	IF Modbus_Slave.rBias_2>rStepBias THEN
		rStepBias:=rStepBias+rStep;
		IF rStepBias>=Modbus_Slave.rBias_2 THEN
			rStepBias:=Modbus_Slave.rBias_2;
		END_IF
	ELSIF Modbus_Slave.rBias_2<rStepBias THEN
		rStepBias:=rStepBias-rStep;
		IF rStepBias<=Modbus_Slave.rBias_2 THEN
			rStepBias:=Modbus_Slave.rBias_2;
		END_IF
	END_IF
	rAuToStepBiasTemp:=0;
ELSIF GVL.bStartTrack AND Axis2Remote.iMode=2 THEN
	Axis2Remote.bStartAutoTrack := TRUE;
	Axis2Remote.rChanU := -AutoTrackingCal.rChanUa;
ELSE
	Axis2Remote.bStartAutoTrack := FALSE;	
	rAuToStepBias:=0;
	rStepBias:=0;
	rAuToStepBiasTemp:=0;
END_IF

// 本控自跟踪
IF GVL.bStartLocalAutoTrack AND Axis2Local.iMode = 4 THEN
	Axis2Local.bStartAutoTrack := TRUE;
	Axis2Local.rChanU := -AutoTrackingCal.rChanUaLocal;
ELSE
	Axis2Local.bStartAutoTrack := FALSE;
END_IF

// =============================================================================
// 段 9: 合成 rPIDCmdPos（注意 AZ_out 为减）→ Az_Ctrl_FB
// =============================================================================
Axis2Remote.rPIDCmdPos:=RealTimePosCal.rInterAzPos+rStepBias+rAuToStepBias+rSearchNextStepTarget-SECURITYCHECK.AZ_out+rAuToStepBiasTemp;

IF Axis2Remote.rPIDCmdPos<-275 THEN
	Axis2Remote.rPIDCmdPos:=-275;
ELSIF Axis2Remote.rPIDCmdPos>275 THEN
	Axis2Remote.rPIDCmdPos:=275;
END_IF

Axis2_Ctrl(sLocal:=Axis2Local, sCtrl:=Axis2Remote, sStatus:=Axis2Status, sVisible:=Axis2Visible, rRealPos:=rFctPosReal_2, rPosLimK:=0.34);

END_PROGRAM

// Device/Application/El_ctrl_1
PROGRAM El_ctrl_1

VAR
    Axis1_Ctrl : El_Ctrl_FB;           // 俯仰轴控制 FB（阶段 4 已注释）
    bRemote2LocalStop : BOOL;          // 远控→本控切换中，需先减速下电
    bLocal2RemoteStop : BOOL;          // 本控→远控切换中，需先减速下电
    Error : INT;                       // 保留
    Axis1Limit_pos : REAL;             // 硬限位上限 180°
    Axis1Limit_Neg : REAL;             // 硬限位下限 93°
    bRTriger : Standard.R_TRIG;        // bLocalCtrl 上升沿（切到本控）
    bFTriger : Standard.F_TRIG;        // bLocalCtrl 下降沿（切到远控）
    Stop1_Count : INT;                 // 低速持续计数（用于判定已停稳）
    bStop_1 : BOOL;                    // TRUE=俯仰轴已停稳（|v|<0.035 持续>1s）
    rPosModeStepBias : LREAL;          // 保留/指向模式步进偏置
    rPosModeStep : LREAL;
    rStepBiasMax : LREAL;
    rStepBias : LREAL;                 // Modbus 下发的手动偏置，逐步逼近 rBias_1
    rStep : LREAL;                     // rStepBias 每拍变化步长
    rAuToStepBias : LREAL;             // 自跟踪累积拉偏 (deg)
    rAuToStepBiasTemp : LREAL;         // 自跟踪瞬时拉偏分量
    rAutoStep : LREAL;                 // 关闭自跟踪后 rAuToStepBias 归零步长
    TbAutoTrigger : Standard.F_TRIG;
    RbAutoTrigger : Standard.R_TRIG;
    rAutoTrackingBiasMax : LREAL;      // 自跟踪拉偏上限
    rLocalInitPosModeSpeed : REAL;
    rRemoteInitPosModeSpeed : REAL;
    iCountOffAuto : INT;
    iCasePBAutoTrack : INT;
    rKAuToStepBias : LREAL;            // 自跟踪拉偏增益系数
    agcmaxsearch_tb : AGCMaxSearch_PB_1;  // 指向模式(mode2) AGC 峰值搜索
    rSearchNextStepTarget_tb : REAL;      // 指向模式搜索输出偏置
    agcmaxsearch_pb : AGCMaxSearch_PB_1;  // 程引模式(mode4) AGC 峰值搜索
    rElthreshold : REAL;               // 俯仰角阈值：仅高于此值才在程引下做 AGC 搜索
    toN1 : Standard.Ton;
    ttime1 : TIME;
    bstartagcmaxsearch : BOOL;
    rSearchNextStepTarget : REAL;      // 程引模式 AGC 搜索输出偏置
    rMaxPosTest : REAL;                // AGC 搜索调试：峰值位置
END_VAR


(*==============================================================================
  PRG: El_ctrl_1（俯仰轴 El 顶层程序）
  任务: Canopen 10ms
  作用:
    1. 读 CANopen 反馈 → 换算实际速度/位置 (rFctVelReal_1 / rFctPosReal_1)
    2. 组装 Axis1Status（故障、使能、运动中等）
    3. 远/本控切换保护、自跟踪拉偏、AGC 峰值搜索
    4. 合成 PID 目标位置 rPIDCmdPos → 调用 El_Ctrl_FB
  数据流:
    Modbus/上位机 → Axis1Remote（在 Modbus_Slave 等处赋值）
    RealTimePosCal.rInterElPos + 各类偏置 → rPIDCmdPos → El_Ctrl_FB → GVL.diEl*
==============================================================================*)




(* 远控参量曾在此从 Modbus_Slave 直赋，现改由 Modbus_Slave 程序统一写入 Axis1Remote *)

// =============================================================================
// 段 1: 驱动状态字 → Axis1Status（供 El_Ctrl_FB 与 HMI 使用）
// DS402 状态: bit0/1/2 同时为 1 表示 Operation Enabled（伺服已使能）
// =============================================================================
Axis1Status.Error := GVL.bElStsBit3;
Axis1Status.ErrorID := GVL.eElErrorcode;
Axis1Status.bServo_Enable := GVL.bElStsBit0 AND GVL.bElStsBit1 AND GVL.bElStsBit2;
Axis1Status.bBrake := NOT (GVL.bElStsBit0 AND GVL.bElStsBit1 AND GVL.bElStsBit2);
Axis1Status.Disabled := NOT (GVL.bElStsBit0 AND GVL.bElStsBit1 AND GVL.bElStsBit2);
// 软限位写入命令结构体（与下面硬限位 93~180 一致）
Axis1Remote.rSoft_limit_Negative:=93;Axis1Remote.rSoft_limit_Postive:=180;
Axis1Local.rSoft_limit_Negative:=93;Axis1Local.rSoft_limit_Postive:=180;

// =============================================================================
// 段 2: CANopen 反馈 → 实际速度/位置（deg, deg/s）
// 公式: 物理量 = diActXxx / 524288 × 360；俯仰另加 Modbus 标定偏移 lrElOffset
// =============================================================================
rFctVelReal_1:=DINT_TO_REAL(diElActVel)/524288.0*360.0;
rFctPosReal_1:=DINT_TO_REAL(diElActPos)/524288.0*360.0 + modbus_slave.lrElOffset;

// =============================================================================
// 段 3: 指向命令硬限位（远控/本控 rPosCmd 钳位到 93°~180°）
// =============================================================================
Axis1Limit_pos:=180;
Axis1Limit_Neg:=93;
IF Axis1Remote.rPosCmd>Axis1Limit_pos THEN
	Axis1Remote.rPosCmd:=180;
ELSIF Axis1Remote.rPosCmd<Axis1Limit_Neg THEN
	 Axis1Remote.rPosCmd:=93;  
END_IF

IF Axis1Local.rPosCmd>Axis1Limit_pos THEN
	Axis1Local.rPosCmd:=180;
ELSIF Axis1Local.rPosCmd<Axis1Limit_Neg THEN
	 Axis1Local.rPosCmd:=93;  
END_IF

// =============================================================================
// 段 4: 停稳判定 → Axis1Status.Moving
// |速度|<0.035°/s 连续 100 拍(约1s) 认为停稳；bStop_1=TRUE → Moving=FALSE
// =============================================================================
IF  ABS(rFctVelReal_1)<0.035 THEN
	Stop1_Count:=Stop1_Count+1;
	IF Stop1_Count>100 THEN
		Stop1_Count:=101;
		bStop_1:=TRUE;;
	END_IF
ELSE
	Stop1_Count:=0;
	bStop_1:=FALSE;
END_IF
Axis1Status.Moving := NOT bStop_1;

// =============================================================================
// 段 5: PID 使能 — 仅指向(2)与程引(4)模式需要位置环
// =============================================================================
IF Axis1Remote.iMode=2 OR Axis1Remote.iMode=4 THEN
	Axis1Remote.bPIDEnable:=TRUE;
ELSE
	Axis1Remote.bPIDEnable:=FALSE;
END_IF

// =============================================================================
// 段 6: 远控 ↔ 本控 切换保护（GVL.bLocalCtrl）
// 切换瞬间若伺服仍使能 → 置切换标志 → 强制 mode=7(halt) 减速
// 停稳且下电完成后 → mode=0，清除标志
// =============================================================================
bRTriger(CLK:=GVL.bLocalCtrl);
bFTriger(CLK:=GVL.bLocalCtrl);

// 远控 → 本控（bLocalCtrl 上升沿）
IF Axis1Status.bServo_Enable AND (bRTriger.Q ) THEN//如果速度不为0且本控发生切换，则减速停止标识为True
	bRemote2LocalStop:=TRUE;
END_IF
IF bRemote2LocalStop  THEN //若减速停止标识符为True 
	
	IF  bStop_1=TRUE THEN//且电机速度不为0 开始减速 减速完成后下使能，下使能完成后复位标识符复位
		Axis1Local.iMode:=0;
		Axis1Remote.iMode:=0;
		IF Axis1Status.bServo_Enable=FALSE THEN
			bRemote2LocalStop:=FALSE;
		END_IF
	ELSE
		Axis1Local.iMode:=7;
		Axis1Remote.iMode:=7;
	END_IF
END_IF

// 本控 → 远控（bLocalCtrl 下降沿）
IF Axis1Status.bServo_Enable AND (bFTriger.Q ) THEN//如果速度不为0且本控发生切换，则减速停止标识为True
	bLocal2RemoteStop:=TRUE;
END_IF
IF bLocal2RemoteStop  THEN //若减速停止标识符为True 
	
	IF  bStop_1=TRUE THEN//且电机速度不为0 开始减速 减速完成后下使能，下使能完成后复位标识符复位
		Axis1Local.iMode:=0;
		Axis1Remote.iMode:=0;
		IF Axis1Status.bServo_Enable=FALSE THEN
			bLocal2RemoteStop:=FALSE;
		END_IF
	ELSE
		Axis1Remote.iMode:=7;
		Axis1Local.iMode:=7;
	END_IF
END_IF

// =============================================================================
// 段 7: AGC 峰值搜索（与方位 Az_ctrl_1 协同，bstartSearchEl 由方位触发）
// mode2: 插值目标 = rPosCmd；mode4: 插值目标 = RealTimePosCal.rInterElPos
// 仅当俯仰高于 rElthreshold（相对水平）且在程引下才在 mode4 启用搜索
// =============================================================================
IF Axis1Remote.iMode=2 THEN
			IF GVL.Chan1AGC>=(GVL.Chanthreshold-0.1) THEN
					agcmaxsearch_pb(bstart:=Az_ctrl_1.agcmaxsearch_tb.bSucess,rAGCNow:=GVL.Chan1AGC,btrig:=Az_ctrl_1.bstartSearchEl,
						rCurrentPos:=rFctPosReal_1,rInterPos:=Axis1Remote.rPosCmd,
				rStepBiasNow:=rStepBias,bAutoTracking:=GVL.bStartTrack,bStop:=FALSE,
				rStepBias=>rSearchNextStepTarget_tb,rAGCMaxBias=>rMaxPosTest,bSucess=>);
			ELSE
				bstartagcmaxsearch:=FALSE;
				agcmaxsearch_pb(bstart:=Az_ctrl_1.agcmaxsearch_tb.bSucess,rAGCNow:=GVL.Chan1AGC,btrig:=Az_ctrl_1.bstartSearchEl,
				rCurrentPos:=rFctPosReal_1,rInterPos:=Axis1Remote.rPosCmd,
				rStepBiasNow:=rStepBias,bAutoTracking:=GVL.bStartTrack,bStop:=FALSE,
				rStepBias=>rSearchNextStepTarget_tb,rAGCMaxBias=>rMaxPosTest,bSucess=>);
			END_IF
		ELSIF Axis1Remote.iMode=4 AND rFctPosReal_1-90>rElthreshold  THEN
			IF GVL.Chan1AGC>=(GVL.Chanthreshold-0.1) THEN
					agcmaxsearch_pb(bstart:=Az_ctrl_1.agcmaxsearch_pb.bSucess,rAGCNow:=GVL.Chan1AGC,btrig:=Az_ctrl_1.bstartSearchEl,
						rCurrentPos:=rFctPosReal_1,rInterPos:=RealTimePosCal.rInterElPos,
				rStepBiasNow:=rStepBias,bAutoTracking:=GVL.bStartTrack,bStop:=FALSE,
				rStepBias=>rSearchNextStepTarget,rAGCMaxBias=>rMaxPosTest,bSucess=>);
			ELSE
				bstartagcmaxsearch:=FALSE;
				agcmaxsearch_pb(bstart:=Az_ctrl_1.agcmaxsearch_pb.bSucess,rAGCNow:=GVL.Chan1AGC,btrig:=Az_ctrl_1.bstartSearchEl,
				rCurrentPos:=rFctPosReal_1,rInterPos:=RealTimePosCal.rInterElPos,
				rStepBiasNow:=rStepBias,bAutoTracking:=GVL.bStartTrack,bStop:=FALSE,
				rStepBias=>rSearchNextStepTarget,rAGCMaxBias=>rMaxPosTest,bSucess=>);
			END_IF
		ELSIF Axis1Remote.iMode =0  OR Axis1Remote.iMode =7 THEN
			bstartagcmaxsearch:=FALSE;
			agcmaxsearch_pb(bstart:=Az_ctrl_1.agcmaxsearch_pb.bSucess,rAGCNow:=GVL.Chan1AGC,btrig:=Az_ctrl_1.bstartSearchEl,
			rCurrentPos:=rFctPosReal_1,rInterPos:=RealTimePosCal.rInterElPos,	
			rStepBiasNow:=rStepBias,bAutoTracking:=GVL.bStartTrack,bStop:=FALSE,
			rStepBias=>rSearchNextStepTarget,rAGCMaxBias=>rMaxPosTest,bSucess=>);
		END_IF

// =============================================================================
// 段 8: 自跟踪拉偏（远控）
// mode4+程引: 用 AutoTrackingCal.rChanUe 累积 rAuToStepBias（限幅）
// mode2+指向: 直接用 rChanU 作 PID 目标增量（在 El_Ctrl_FB 内 rChanU+位置）
// 关跟踪: rAuToStepBias 渐零，rStepBias 渐近 Modbus_Slave.rBias_1
// =============================================================================
IF GVL.bStartTrack AND Axis1Remote.iMode=4 THEN
	Axis1Remote.bStartAutoTrack := TRUE;
	IF rAuToStepBias > rAutoTrackingBiasMax THEN
		rAuToStepBias := rAutoTrackingBiasMax;
	ELSIF rAuToStepBias < -rAutoTrackingBiasMax THEN
		rAuToStepBias := -rAutoTrackingBiasMax;
	ELSE
		rAuToStepBiasTemp:=0.02*AutoTrackingCal.rDirSenFac*AutoTrackingCal.rChanUe;
		rAuToStepBias:=rAuToStepBias+AutoTrackingCal.rDirSenFac*rKAuToStepBias*AutoTrackingCal.rChanUe/1000.0;
	END_IF
ELSIF NOT GVL.bStartTrack AND Axis1Remote.iMode=4 THEN
	IF 	rAuToStepBias>0 THEN//关闭自跟踪后自跟踪拉偏量逐渐归0
		rAuToStepBias:=rAuToStepBias-rAutoStep;
	ELSIF rAuToStepBias<0 THEN
		rAuToStepBias:=rAuToStepBias+rAutoStep;
	ELSE
		rAuToStepBias:=0;
	END_IF
	
	IF Modbus_Slave.rBias_1>rStepBias THEN
		rStepBias:=rStepBias+rStep;
		IF rStepBias>=Modbus_Slave.rBias_1 THEN
			rStepBias:=Modbus_Slave.rBias_1;
		END_IF
	ELSIF Modbus_Slave.rBias_1<rStepBias THEN
		rStepBias:=rStepBias-rStep;
		IF rStepBias<=Modbus_Slave.rBias_1 THEN
			rStepBias:=Modbus_Slave.rBias_1;
		END_IF
	END_IF
	rAuToStepBiasTemp:=0;
ELSIF GVL.bStartTrack AND Axis1Remote.iMode=2 THEN
	Axis1Remote.bStartAutoTrack := TRUE;
	Axis1Remote.rChanU := AutoTrackingCal.rChanUe;
ELSE
	Axis1Remote.bStartAutoTrack := FALSE;	
	rAuToStepBias:=0;
	rStepBias:=0;
	rAuToStepBiasTemp:=0;
END_IF

// 本控自跟踪（仅程引 mode4）
IF GVL.bStartLocalAutoTrack AND Axis1Local.iMode = 4 THEN
	Axis1Local.bStartAutoTrack := TRUE;
	Axis1Local.rChanU := AutoTrackingCal.rChanUeLocal;
ELSE
	Axis1Local.bStartAutoTrack := FALSE;
END_IF

// =============================================================================
// 段 9: 合成 PID 目标位置并限位 → 调用 El_Ctrl_FB
// rPIDCmdPos = 程引插值 + 手动偏置 + 自跟踪偏置 + AGC搜索偏置 + 安全检查偏置
// =============================================================================
Axis1Remote.rPIDCmdPos:=RealTimePosCal.rInterElPos+rStepBias+rAuToStepBias+rSearchNextStepTarget+SECURITYCHECK.el_out+rAuToStepBiasTemp;
IF Axis1Remote.rPIDCmdPos<93 THEN
	Axis1Remote.rPIDCmdPos:=93;
ELSIF Axis1Remote.rPIDCmdPos>180 THEN
	Axis1Remote.rPIDCmdPos:=180;
END_IF

Axis1_Ctrl(sLocal:=Axis1Local, sCtrl:=Axis1Remote, sStatus:=Axis1Status, sVisible:=Axis1Visible, rRealPos:=rFctPosReal_1, rPosLimK:=0.34);

END_PROGRAM

// Device/Application/PID
FUNCTION_BLOCK PID
VAR_INPUT
    rTarget : REAL;              // 目标位置 (deg)
    rFeedback : REAL;            // 实际位置反馈 (deg)
    rPosLimPositive : LREAL;     // 软限位正限 (deg)，超出则输出清零
    rPosLimNegative : LREAL;     // 软限位负限 (deg)
    rKp : REAL;                  // 比例系数
    rKi : REAL;                  // 积分系数
    rKd : REAL;                  // 微分系数（当前逻辑未实际使用）
    iThreshold : INT;            // 积分开启阈值 (deg)；-1 = 始终开积分
    bPIDEnable : BOOL;           // PID 使能，FALSE 时各项清零
    rVelLim : LREAL;             // 输出速度限幅 (deg/s)
END_VAR

VAR_OUTPUT
    rPIDOutput : LREAL;          // PID 输出速度 (deg/s)，写到 diXxTargetVel 前换算
    rPIDtrace : LREAL;           // 调试/显示用，与 rPIDOutput 相同
END_VAR
VAR
    rLastError : LREAL;          // 上一拍误差（当前版本未使用微分，保留备用）
    rErrorNow : LREAL;           // 当前误差 = rTarget - rFeedback
    rIntegralNew : LREAL;        // 积分累计量
    rDerivativeNew : LREAL;      // 微分项（未使用）
    rDelta : LREAL;              // 备用
    rProportionNew : LREAL;      // 比例项 = rErrorNow
END_VAR


(*==============================================================================
  FB: PID（位置环速度输出 PID）
  任务: Canopen 10ms（由 *_Ctrl_FB 调用）
  作用: 输入目标位置与实际位置，输出速度指令（deg/s）
  算法: 比例 + 条件积分（误差小于阈值才累积），无微分
  使用者: El_Ctrl_FB / Az_Ctrl_FB / Ti_Ctrl_FB 中的 VelPID_1/2/3
==============================================================================*)

// ----- 段：PID 使能入口 -----
IF (bPIDEnable>0) THEN //如果PID使能
	IF rTarget=rFeedback THEN
		rPIDOutput:=0;	               // 目标=反馈，输出为 0
	ELSE
	
		rErrorNow:=rTarget-rFeedback;  //计算当前误差 en
		rProportionNew:=rErrorNow;     //比例项

		// ----- 段：条件积分（仅在软限位内、误差小于阈值时才累积）-----
		IF rFeedback>rPosLimNegative AND rFeedback<rPosLimPositive THEN //若在软限位之内，工作时开启积分项
			IF (ABS(rTarget-rFeedback)<iThreshold) THEN//位置差小于积分阈值
				rIntegralNew:= rIntegralNew+rErrorNow; //积分项
			ELSE
				rIntegralNew:=0;
			END_IF;
		ELSE //不在软限位范围内,则积分项为0
			rIntegralNew:=0;
		END_IF

		// ----- 段：PID 求和输出 -----
		rPIDOutPut:=rKp*rProportionNew+rKi*rIntegralNew;
		rPIDtrace:=rKp*rProportionNew+rKi*rIntegralNew;

		// ----- 段：速度限幅（双向） -----
		IF rPIDOutput<(-rVelLim) THEN
			rPIDOutput:=-rVelLim;
		ELSIF rPIDOutput>rVelLim THEN
			rPIDOutput:=rVelLim;
		END_IF
		
		// ----- 段：超软限位时强制输出清零，防止继续向限位方向运动 -----
		IF rFeedback>rPosLimPositive AND rPIDOutput>0 THEN 
			rPIDOutput:=0;
		END_IF
		IF rFeedback<rPosLimNegative AND rPIDOutput<0 THEN
			rPIDOutput:=0;
		END_IF
		
		rLastError:=rErrorNow;//将当前误差赋值给上一次误差
		
	END_IF
ELSE//非使能清零PID各项
	rProportionNew:=0.0;
	rIntegralNew:=0.0;
	rPIDOutput:=0.0;
END_IF

END_FUNCTION_BLOCK

// Device/Application/El_Ctrl_FB
FUNCTION_BLOCK El_Ctrl_FB

VAR_INPUT
    sLocal : AxisCrtlStruct;     // 本控命令结构体（来自本地操作面板/GVL.sXxLocal）
    sCtrl : AxisCrtlStruct;      // 远控命令结构体（来自 Modbus/上位机/GVL.sXxCtrl）
    sStatus : AxisStatus;        // 轴状态（Disabled/Moving/Error 等标志）
    sVisible : AxisVisible;      // HMI 可视化相关（此 FB 内部未直接使用）
    rRealPos : REAL;             // 编码器实际位置 (deg)，即 GVL.rFctPosReal_X
    rPosLimK : REAL;             // 备用限位系数（当前逻辑未使用）
END_VAR

VAR_OUTPUT
    logicError : INT;            // 逻辑错误码（保留，当前未赋值）
END_VAR

VAR
    VelPID_1 : PID;              // 位置模式（positionMode）用普通 PID
    VelPID_2 : PID;              // 本控位置模式（programBootMode 本控）用普通 PID
    VelPID_3 : PID;              // 保留（已被 vpid1 替代，代码中注释掉）
    vpid1 : vpid;                // 变增益 PID，用于 programBootMode 远控/自跟踪
    TON_0 : TON;                 // 延时 1s，错误时判断 stop0 是否超时
    bTick : BOOL;                // stop0 超时后置位，触发强制下电
    tr : BOOL;                   // 心跳错误正在处理中标志（防止重入）
    icount1 : INT;               // 心跳恢复计数器（等 101 拍 ≈ 1s 后清 bit7）
    icount2 : INT;               // 清 bit7 后再等 101 拍才结束保护
    icount3 : INT;               // 备用
    bfin1 : BOOL;                // icount1 到达后置位，触发 icount2 阶段
    bfin2 : BOOL;                // 保留
    istate : INT;                // 上电序列状态机（0→1→2）
    icount : INT;                // 上电序列各步骤等待计数（20 拍 = 200ms）
END_VAR


(*==============================================================================
  FB: El_Ctrl_FB（俯仰轴 Elevation 控制功能块）
  任务: Canopen 10ms（周期调用）
  作用:
    - 根据 sCtrl/sLocal 的 iMode，产生对应 CANopen 速度/控制字写入
    - 封装上/下电序列、软限位保护、CANopen 错误码自动恢复、心跳丢失处理
    - 内部调用 PID / vpid 进行位置→速度的闭环换算
  输入: sCtrl（远控命令结构体）、sLocal（本控命令结构体）
        sStatus（轴状态）、rRealPos（编码器实际角度）
  输出: 直接写 GVL.diElTargetVel / diElTargetAcc / diElTargetDec 及控制字位

  速度换算公式（通用）:
    diXxTargetVel [inc/s] = deg/s × 524288 / 360
    其中 524288 = 2^19（CANopen 电机编码器增量/转，具体由电机参数决定）
==============================================================================*)


// =============================================================================
// 段 A: 全局复位 — 轴停止或下电时清 bit8（快速停止位）
// bit8=1 激活快速停止，bit8=0 正常运行
// =============================================================================
IF sStatus.Disabled OR (NOT sStatus.Moving) THEN
	bElCtrlBit8 := FALSE;
END_IF

// =============================================================================
// 段 B: 错误复位（由 HMI 或 Modbus 写 bError_Reset）
// 将两个命令结构体模式设为 reset(6)，清 Error_code
// =============================================================================
IF GVL.bError_Reset THEN
	sCtrl.iMode:=6;
	sLocal.iMode:=6;
	GVL.Error_code:=0;
END_IF
IF GVL.Error_code =0 THEN
	GVL.bError_Reset:=FALSE;
END_IF

// =============================================================================
// 段 C: CANopen 心跳超时错误（错误码 0x8130）自动恢复序列
// 步骤: 设 bit7(故障复位位) → 等 101 拍 → 清 bit7 → 再等 101 拍 → 结束
// 期间同时下电（清控制字 bit0~3），待驱动自愈后再由上层重新上电
// =============================================================================
IF GVL.eElErrorcode = 16#8130 AND NOT tr THEN
	GVL.bElCtrlBit7 := TRUE;  // 触发驱动故障复位
	tr:=TRUE;
	istate:=0;
	icount:=0;
	// 写入下电控制字
	GVL.bElCtrlBit3 := FALSE;
	GVL.bElCtrlBit0 := FALSE;
	GVL.bElCtrlBit1 := FALSE;
	GVL.bElCtrlBit2 := FALSE;	
END_IF
IF tr THEN
	icount1 := icount1 + 1;
END_IF
IF icount1 > 101 THEN     // 约 1s（10ms × 101）后清故障复位位
	icount1 := 0;
	tr := FALSE;
	GVL.bElCtrlBit7 := FALSE;
	bfin1 := TRUE;
END_IF
IF bfin1 THEN             // 再等 1s 让驱动彻底稳定
	icount2 := icount2 + 1;
END_IF
IF icount2 > 101 THEN
	bfin1 := FALSE;
	icount2 := 0;
END_IF

// =============================================================================
// 段 D: 主控制逻辑
// 条件: 无全局错误 AND 无驱动错误 AND 不在心跳恢复序列中
// =============================================================================
IF GVL.Error_code=0 AND GVL.eElErrorcode = 0 AND NOT GVL.bElCtrlBit7  AND NOT tr AND NOT bfin1 AND NOT bfin2 THEN

	// =========== 远控分支（bLocalCtrl=FALSE） ===========
	IF GVL.bLocalCtrl=FALSE THEN //远控
		IF sCtrl.iMode <> 1 THEN   // 非上电模式时重置上电状态机
			istate:=0;
			icount:=0;
		END_IF
		CASE sCtrl.iMode OF

			// ----- 模式 0: 下电 -----
			MODES.powerOff: // 下电
				IF NOT sStatus.Disabled THEN
					IF sStatus.Moving THEN // 运动中，先停止运动
						GVL.diElTargetVel := 0;
						bElCtrlBit8 := TRUE;   // 发快速停止
					ELSE
						// 写入下电控制字（bit0~3=0 即断使能）
						GVL.bElCtrlBit3 := FALSE;
						GVL.bElCtrlBit0 := FALSE;
						GVL.bElCtrlBit1 := FALSE;
						GVL.bElCtrlBit2 := FALSE;
					END_IF
				END_IF
				// 注: 下电模式仍持续运行 vpid1，但输出不写到 diElTargetVel
				// 目的是让 vpid1 内部积分不要突变（实际速度已通过控制字停掉）
				vpid1(rKpbase:=1, rKibase:=0.01, rKpMax:=1, rKiMax:=0.01, rVelThreshold:=10,rTarget:=sCtrl.rPIDCmdPos,rFeedback:=rRealPos,rPosLimPositive:=sCtrl.rSoft_limit_Postive,
							rPosLimNegitive:=sCtrl.rSoft_limit_Negative,
								bPIDEnable:=sCtrl.bPIDEnable,rVelLim:=sCtrl.rVel_Limit,rKpScale:=0.02,rKiScale:=0.005,rElPos:=GVL.rFctPosReal_1-90,
								iThrehold:=sCtrl.rPIDThre,rPIDOutDir=>sCtrl.rPIDCmdVel);

			// ----- 模式 1: 上电（三步 CANopen DS402 状态机）-----
			MODES.powerOn:  // 上电
				IF sStatus.Disabled THEN
					GVL.diElTargetVel := 0;
					IF GVL.siElMode <> 3 THEN // 上电时模式默认为3，速度模式
						GVL.siElMode := 3;
					END_IF
					IF siElMode = 3 THEN
						// DS402 上电序列: Shutdown → Switch On → Enable Operation
						// 每步等待 20 拍（200ms）确保驱动应答
						CASE istate OF
							0:  // Shutdown: bit1=1, bit2=1（清故障 + 切换允许）
								GVL.bElCtrlBit1 := TRUE;
								GVL.bElCtrlBit2 := TRUE;
								icount := icount + 1;
								IF icount = 20 THEN
									icount:=0;
									istate:=1;
								END_IF
							1:  // Switch On: bit0=1
								GVL.bElCtrlBit0 := TRUE;
								icount := icount + 1;
								IF icount = 20 THEN
									icount:=0;
									istate:=2;
								END_IF
							2:  // Enable Operation: bit3=1
								GVL.bElCtrlBit3 := TRUE;
						END_CASE
					END_IF
				ELSE
					// 已上电：若还在运动则发快速停止等待停稳
					IF sStatus.Moving THEN
						GVL.diElTargetVel := 0;
						bElCtrlBit8 := TRUE;
					ELSE
						bElCtrlBit8 := FALSE;
					END_IF
				END_IF

			// ----- 模式 2: 指向模式（位置 PID 输出速度，远控）-----
			MODES.positionMode: // 远控指向模式
				IF NOT sStatus.Disabled THEN
					IF sCtrl.bStartAutoTrack THEN
						// 自跟踪模式：误差电压（rChanU）直接作为位置增量指令
						// 即: 目标 = rChanU（deg，来自跟踪接收机） + 当前位置
						VelPID_1(rTarget:=sCtrl.rChanU + rRealPos,
								rFeedback:=rRealPos,
								rPosLimPositive:=sCtrl.rSoft_limit_Postive,
								rPosLimNegative:=sCtrl.rSoft_limit_Negative,
								rVelLim:=sCtrl.rVel_Limit,
								rKp:=1,//自跟踪PI系数3,0.02
								rKi:=0,
								rKd:=0,
								bPIDEnable:=sCtrl.bPIDEnable,
								iThreshold:= -1,   // -1=始终开积分
								rPIDOutput=>sCtrl.rPIDCmdVel);							
					ELSE
						// 指向模式：目标为上位机给定的角度
						VelPID_1(rTarget:=sCtrl.rPosCmd,
							rFeedback:=rRealPos,
							rVelLim:=sCtrl.Pos_Vel,
							rPosLimPositive:=sCtrl.rSoft_limit_Postive,
							rPosLimNegative:=sCtrl.rSoft_limit_Negative,
							rKp:=0.7,//程引PI系数地带：1,0.002  高带：3,0.02
							rKi:=0,
							rKd:=0,
							bPIDEnable:=sCtrl.bPIDEnable,
							iThreshold:=sCtrl.rPIDThre,
							rPIDOutput=>sCtrl.rPIDCmdVel);
					END_IF
					// 将 PID 输出速度(deg/s)换算为 CANopen 速度增量单位写入
					GVL.diElTargetVel := REAL_TO_DINT(sCtrl.rPIDCmdVel * 524288 / 360);
					GVL.diElTargetAcc := REAL_TO_UDINT(9 * 524288 / 360);   //加速度 9 deg/s²
					GVL.diElTargetDec := REAL_TO_UDINT(9 * 524288 / 360);   //减速度
				END_IF

			// ----- 模式 3: 速度模式（手动点动，远控）-----
			MODES.velocityMode://手控速度模式-远控模式
				IF NOT sStatus.Disabled THEN
					// 限幅处理：超过限速则取限速值
					IF ABS(sCtrl.rVelCmd) <= sCtrl.rVel_Limit THEN
						GVL.diElTargetVel := REAL_TO_DINT(sCtrl.rVelCmd * 524288 / 360);
					ELSIF sCtrl.rVelCmd > sCtrl.rVel_Limit THEN
						GVL.diElTargetVel := REAL_TO_DINT(sCtrl.rVel_Limit * 524288 / 360);
					ELSE
						GVL.diElTargetVel := REAL_TO_DINT(-sCtrl.rVel_Limit * 524288 / 360);
					END_IF
					GVL.diElTargetAcc := REAL_TO_UDINT(sCtrl.rAcceleration * 524288 / 360);   //加速度
					GVL.diElTargetDec := REAL_TO_UDINT(sCtrl.rDeceleration * 524288 / 360);   //减速度
				END_IF

			// ----- 模式 4: 程引模式（程序引导/插值跟踪，远控）-----
			// 使用变增益 vpid1，参数来自 PersistentVars（标定可调）
			MODES.programBootMode://PID速度模式-正常模式 程引
				IF NOT sStatus.Disabled THEN
					IF sCtrl.bStartAutoTrack THEN
						// 程引+自跟踪：误差电压叠加到插值目标位置上
						vpid1(rKpbase:=Persistentvars.rElKpBase, rKibase:=Persistentvars.rElKiBase, rKpMax:=Persistentvars.rElKpMax, rKiMax:=Persistentvars.rElKiMax, rVelThreshold:=Persistentvars.rElThre,rTarget:=sCtrl.rPIDCmdPos,rFeedback:=rRealPos,rPosLimPositive:=sCtrl.rSoft_limit_Postive,
							rPosLimNegitive:=sCtrl.rSoft_limit_Negative,
								bPIDEnable:=sCtrl.bPIDEnable,rVelLim:=sCtrl.rVel_Limit,rKpScale:=Persistentvars.rElKpscale,rKiScale:=Persistentvars.rElKiscale,rElPos:=GVL.rFctPosReal_1-90,
								iThrehold:=sCtrl.rPIDThre,rPIDOutDir=>sCtrl.rPIDCmdVel);						
					ELSE
						// 程引不开自跟踪：纯插值位置跟踪
						vpid1(rKpbase:=Persistentvars.rElKpBase, rKibase:=Persistentvars.rElKiBase, rKpMax:=Persistentvars.rElKpMax, rKiMax:=Persistentvars.rElKiMax, rVelThreshold:=Persistentvars.rElThre,rTarget:=sCtrl.rPIDCmdPos,rFeedback:=rRealPos,rPosLimPositive:=sCtrl.rSoft_limit_Postive,
							rPosLimNegitive:=sCtrl.rSoft_limit_Negative,
								bPIDEnable:=sCtrl.bPIDEnable,rVelLim:=sCtrl.rVel_Limit,rKpScale:=Persistentvars.rElKpscale,rKiScale:=Persistentvars.rElKiscale,rElPos:=GVL.rFctPosReal_1-90,
								iThrehold:=sCtrl.rPIDThre,rPIDOutDir=>sCtrl.rPIDCmdVel);
					END_IF
					GVL.diElTargetVel := REAL_TO_DINT(sCtrl.rPIDCmdVel * 524288 / 360);
					GVL.diElTargetAcc := REAL_TO_UDINT(sCtrl.rAcceleration * 524288 / 360);   //加速度
					GVL.diElTargetDec := REAL_TO_UDINT(sCtrl.rDeceleration * 524288 / 360);   //减速度
				END_IF

			// ----- 模式 6: 重置 -----
			MODES.reset://重置
				IF NOT sStatus.Disabled THEN
					IF sStatus.Moving THEN
						GVL.diElTargetVel := 0;
						bElCtrlBit8 := TRUE;
					ELSE
						bElCtrlBit8 := FALSE;
					END_IF
				END_IF

			// ----- 模式 5: 待机（停止运动，保持上电）-----
			MODES.halt://待机
				IF NOT sStatus.Disabled THEN
					IF sStatus.Moving THEN
						GVL.diElTargetVel := 0;
						bElCtrlBit8 := TRUE;
					ELSE
						bElCtrlBit8 := FALSE;
					END_IF
				END_IF
			
		END_CASE

	// =========== 本控分支（bLocalCtrl=TRUE）===========
	ELSE // 本控
		IF sLocal.iMode <> 1 THEN
			istate:=0;
			icount:=0;
		END_IF
		CASE sLocal.iMode OF

			MODES.powerOff: // 下电
				IF NOT sStatus.Disabled THEN
					IF sStatus.Moving THEN // 运动中，先停止运动
						GVL.diElTargetVel := 0;
						bElCtrlBit8 := TRUE;
					ELSE
						// 写入下电控制字
						GVL.bElCtrlBit3 := FALSE;
						GVL.bElCtrlBit0 := FALSE;
						GVL.bElCtrlBit1 := FALSE;
						GVL.bElCtrlBit2 := FALSE;
					END_IF
				END_IF

			MODES.powerOn:  // 上电（与远控相同的三步序列）
				IF sStatus.Disabled THEN
					GVL.diElTargetVel := 0;
					IF GVL.siElMode <> 3 THEN // 上电时模式默认为3，速度模式
						GVL.siElMode := 3;
					END_IF
					IF siElMode = 3 THEN
						CASE istate OF
							0:
								GVL.bElCtrlBit1 := TRUE;
								GVL.bElCtrlBit2 := TRUE;
								icount := icount + 1;
								IF icount = 20 THEN
									icount:=0;
									istate:=1;
								END_IF
							1:
								GVL.bElCtrlBit0 := TRUE;
								icount := icount + 1;
								IF icount = 20 THEN
									icount:=0;
									istate:=2;
								END_IF
							2:
								GVL.bElCtrlBit3 := TRUE;
						END_CASE
					END_IF
				ELSE
					IF sStatus.Moving THEN
						GVL.diElTargetVel := 0;
						bElCtrlBit8 := TRUE;
					ELSE
						bElCtrlBit8 := FALSE;
					END_IF
				END_IF

			MODES.velocityMode://手控速度模式-本控模式
				IF NOT sStatus.Disabled THEN
					IF ABS(sLocal.rVelCmd) <= sLocal.rVel_Limit THEN
						GVL.diElTargetVel := REAL_TO_DINT(sLocal.rVelCmd * 524288 / 360);
					ELSIF sLocal.rVelCmd > sLocal.rVel_Limit THEN
						GVL.diElTargetVel := REAL_TO_DINT(sLocal.rVel_Limit * 524288 / 360);
					ELSE
						GVL.diElTargetVel := REAL_TO_DINT(-sLocal.rVel_Limit * 524288 / 360);
					END_IF
					GVL.diElTargetAcc := REAL_TO_UDINT(sLocal.rAcceleration * 524288 / 360);   //加速度
					GVL.diElTargetDec := REAL_TO_UDINT(sLocal.rDeceleration * 524288 / 360);   //减速度
				END_IF

			MODES.programBootMode://本控位置模式（普通 PID，不用变增益）
				IF NOT sStatus.Disabled THEN
					IF NOT sLocal.bPIDEnable THEN
						GVL.diElTargetVel := 0;							
					ELSE
						IF NOT slocal.bStartAutoTrack THEN
							// 纯位置跟踪 PID
							 VelPID_2(rTarget:=sLocal.rPosCmd,
									 rFeedback:=rRealPos,
									 rPosLimPositive:=sLocal.rSoft_limit_Postive,//软限位
									 rPosLimNegative:=sLocal.rSoft_limit_Negative,
									 rKp:=0.7,
									 rKi:=0,
									 rKd:=0,
									 iThreshold:=sLocal.rPIDThre,
									 bPIDEnable:=sLocal.bPIDEnable,
									 rVelLim:=sLocal.Pos_Vel,
									 rPIDOutput=>sLocal.rPIDCmdVel);//普通PID
						ELSE
							// 本控自跟踪：误差电压叠加
							 VelPID_2(rTarget:=sLocal.rChanU + rRealPos,
								rFeedback:=rRealPos,
								rPosLimPositive:=sLocal.rSoft_limit_Postive,
								rPosLimNegative:=sLocal.rSoft_limit_Negative,
								rVelLim:=sLocal.rVel_Limit,
								rKp:=1,//自跟踪PI系数3,0.02
								rKi:=0,
								rKd:=0,
								bPIDEnable:=sLocal.bPIDEnable,
								iThreshold:= -1,
								rPIDOutput=>sLocal.rPIDCmdVel);
						END_IF
						
					END_IF
					GVL.diElTargetVel := REAL_TO_DINT(sLocal.rPIDCmdVel * 524288 / 360);
					GVL.diElTargetAcc := REAL_TO_UDINT(9 * 524288 / 360);   //加速度
					GVL.diElTargetDec := REAL_TO_UDINT(9 * 524288 / 360);   //减速度
				END_IF

			MODES.reset://重置
			// 是否需要
			MODES.halt://待机
				IF NOT sStatus.Disabled THEN
					IF sStatus.Moving THEN
						GVL.diElTargetVel := 0;
						bElCtrlBit8 := TRUE;
					ELSE
						bElCtrlBit8 := FALSE;
					END_IF
				END_IF
			
		END_CASE
	END_IF

// =============================================================================
// 段 E: 全局错误时强制停轴（Error_code≠0 但驱动本身无错，属于上层逻辑错误）
// 发快速停止，超时 1s 后强制下电
// =============================================================================
ELSIF GVL.Error_code<>0 AND GVL.eElErrorcode = 0 AND NOT GVL.bElCtrlBit7  AND NOT tr AND NOT bfin1 AND NOT bfin2 THEN
	// 出现错误，轴停止运动
	GVL.diElTargetVel := 0;
	bElCtrlBit8 := TRUE;
	TON_0(IN:=bElCtrlBit8,PT:=T#1S,Q=>,ET=>);//判断stop0执行是否超时,若超时强制下电（手动复位）
	IF TON_0.Q THEN
		bTick:=TRUE;
	END_IF
	IF bTick AND sStatus.Moving THEN // 超时强制下电
		// 写入下电控制字
		GVL.bElCtrlBit3 := FALSE;
		GVL.bElCtrlBit0 := FALSE;
		GVL.bElCtrlBit1 := FALSE;
		GVL.bElCtrlBit2 := FALSE;
	END_IF
END_IF

END_FUNCTION_BLOCK

// Device/Application/vpid
FUNCTION_BLOCK vpid
VAR_INPUT
    rTarget : REAL;              // 目标位置 (deg)
    rFeedback : REAL;            // 实际位置 (deg)
    rPosLimPositive : LREAL;     // 软限位正限 (deg)
    rPosLimNegitive : LREAL;     // 软限位负限 (deg)（注：原拼写 Negitive，勿改）
    rKpBase : REAL;              // Kp 基础值（低速/低角度区）
    rKiBase : REAL;              // Ki 基础值
    rVelThreshold : LREAL;       // 增益切换阈值：rElPos 超过此值开始叠加增益
    rKpScale : REAL;             // Kp 随角度的线性缩放斜率
    rKiScale : REAL;             // Ki 随角度的线性缩放斜率
    iThrehold : INT;             // 积分开启的误差阈值 (deg)
    bPIDEnable : BOOL;           // PID 使能
    rVelLim : LREAL;             // 输出速度限幅 (deg/s)
    rKpMax : REAL;               // Kp 上限
    rKiMax : REAL;               // Ki 上限
    rElPos : REAL;               // 当前俯仰实际角度，用于动态调整增益（GVL.rFctPosReal_1-90）
END_VAR

VAR_OUTPUT
    rPIDOutput : LREAL;          // 不带限位检查的原始输出（内部过渡量）
    rPIDOutDir : LREAL;          // 最终输出速度 (deg/s)，写 diXxTargetVel 前换算
END_VAR

VAR
    rLastFeedback : LREAL;       // 备用（当前版本已注释掉速度计算）
    rErrorNow : LREAL;           // 当前位置误差
    rIntegralNew : LREAL;        // 积分累计
    rDelta : LREAL;              // 备用
    rProportionNew : LREAL;      // 比例项 = rErrorNow
    rSpeed : REAL;               // 备用（速度自适应已注释）
    rKp : REAL;                  // 当前实际 Kp（动态跟踪 rKpTarget）
    rKi : REAL;                  // 当前实际 Ki
    rInterValueNow : LREAL;      // 备用（插值速度，已注释）
    rInterValueLast : LREAL;     // 备用
    rStep : LREAL;               // Kp/Ki 每拍变化步长（防止突变）
    rKpTarget : REAL;            // 目标 Kp（由 rElPos 计算）
    rKiTarget : REAL;            // 目标 Ki
END_VAR

(*==============================================================================
  FB: vpid（变增益自适应 PID）
  任务: Canopen 10ms（由 El_Ctrl_FB / Az_Ctrl_FB 在 programBootMode 下调用）
  作用: 与 PID 相似，但 Kp/Ki 根据当前俯仰角（rElPos）动态调整
        俯仰角越大（天线仰角越高），摩擦力和惯量变化大，需更高增益
  与 PID 的区别:
    - 输入参数带 Kp/Ki 基础值、缩放因子、最大值
    - 内部按 rElPos > rVelThreshold 时线性增加 Kp/Ki
    - 输出走 rPIDOutDir（方向输出）而非 rPIDOutput
  来源参数: PersistentVars.rXxKpBase/rXxKiBase 等（掉电保持，可由 HMI/Modbus 标定）
==============================================================================*)

// ----- 段：PID 使能入口 -----
IF (bPIDEnable) THEN // 如果PID使能
    IF rTarget = rFeedback THEN
        rPIDOutDir := 0;    
    ELSE
        rErrorNow := rTarget - rFeedback; // 计算当前误差
        rProportionNew := rErrorNow;      // 比例项
		
		// ----- 段：根据俯仰角动态计算目标 Kp/Ki -----
		// rElPos = 当前俯仰角 - 90，即相对水平的仰角
		// 当仰角 > rVelThreshold 时，增益线性增加
		IF rElPos > rVelThreshold THEN
			rKpTarget := rKpBase + rKpScale * (rElPos - rVelThreshold);
			rKiTarget := rKiBase + rKiScale * (rElPos - rVelThreshold);
		ELSE
			rKpTarget := rKpBase;
			rKiTarget := rKiBase;
		END_IF
        // ----- 段：Kp/Ki 上限保护 -----
        IF rKpTarget > rKpMax THEN
			rKpTarget := rKpMax;
		END_IF
		IF rKiTarget > rKiMax THEN
			rKiTarget := rKiMax;
		END_IF
		
		// ----- 段：Kp/Ki 平滑追踪目标值（rStep 步进，防增益突变抖动）-----
		IF rKp<=rKpTarget THEN
			rKp:=rKp+rStep;
		ELSE
			rKp:=rKp-rStep;
		END_IF
		IF rKi<=rKiTarget THEN
			rKi:=rKi+(rKiScale/rKpScale)*rStep;
		ELSE
			rKi:=rKi-(rKiScale/rKpScale)*rStep;
		END_IF
	END_IF

        // ----- 段：条件积分（与 PID 相同逻辑）-----
        IF rFeedback > rPosLimNegitive AND rFeedback < rPosLimPositive THEN // 若在软限位之内，工作时开启积分项
            IF (ABS(rTarget - rFeedback) < iThrehold) THEN // 位置差小于积分阈值
                rIntegralNew := rIntegralNew + rErrorNow;  // 积分项
            ELSE
                rIntegralNew := rIntegralNew;  // 积分项
            END_IF;
        ELSE // 不在软限位范围内，则积分项为0
            rIntegralNew := 0;
        END_IF
        (*
        // 防止目标位置与当前位置偏差过大，导致比例项输出太大，引起震动
        IF rKp * rProportionNew > 2 THEN
            rPIDOutput := 2;
        ELSIF rKp * rProportionNew < -2 THEN
            rPIDOutput := -2;
        ELSE
            rPIDOutput := rKp * rProportionNew + rKi * rIntegralNew / 1000.0; // 由于需求积分项过小，因此积分系数在接口数据上除1000
        END_IF
        *)
		rPIDOutput := rKp * rProportionNew + rKi * rIntegralNew; // 由于需求积分项过小，因此积分系数在接口数据上除1000
        // 根据方向设置输出
        IF rPIDOutput < 0 THEN
            rPIDOutDir := rPIDOutput;
        ELSE
            rPIDOutDir := rPIDOutput;
        END_IF
        
        // ----- 段：速度限幅 -----
        IF (ABS(rPIDOutDir) > rVelLim) THEN
            IF rPIDOutDir < (-rVelLim) THEN
                rPIDOutDir := -rVelLim;
            ELSIF rPIDOutDir > rVelLim THEN
                rPIDOutDir := rVelLim;
            END_IF
        END_IF
        
        // ----- 段：超软限位时强制输出清零 -----
        IF rFeedback > rPosLimPositive AND rPIDOutDir > 0  THEN
            rPIDOutDir := 0;
        END_IF
        IF rFeedback < rPosLimNegitive AND rPIDOutDir <= 0 THEN
            rPIDOutDir := 0;
        END_IF
        
        //rLastFeedback := rFeedback; // 将当前反馈值赋值给上一次反馈值
		//rInterValueLast := rInterValueNow; // 将当前插值位置值赋值给上一次

ELSE // 非使能清零PID各项
    rProportionNew := 0.0;
    rIntegralNew := 0.0;
    rPIDOutDir := 0.0;
    rPIDOutput := 0.0;
END_IF

END_FUNCTION_BLOCK

// Device/Application/Az_Ctrl_FB
FUNCTION_BLOCK Az_Ctrl_FB

VAR_INPUT
    sLocal : AxisCrtlStruct;     // 本控命令结构体
    sCtrl : AxisCrtlStruct;      // 远控命令结构体
    sStatus : AxisStatus;        // 轴状态
    sVisible : AxisVisible;      // HMI 可视化（此 FB 未直接使用）
    rRealPos : REAL;             // 编码器实际位置 (deg)
    rPosLimK : REAL;             // 备用限位系数
END_VAR

VAR_OUTPUT
    logicError : INT;            // 保留
END_VAR

VAR
    VelPID_1 : PID;              // positionMode 用
    VelPID_2 : PID;              // 本控 programBootMode 用
    VelPID_3 : PID;              // 保留（已被 vpid1 替代）
    vpid1 : vpid;                // 变增益 PID，programBootMode 远控
    TON_0 : TON;                 // 超时 1s 强制下电计时器
    bTick : BOOL;                // stop0 超时标志
    tr : BOOL;                   // 心跳恢复进行中标志
    icount1 : INT;               // 心跳恢复计数器1
    icount2 : INT;               // 心跳恢复计数器2
    icount3 : INT;               // 备用
    bfin1 : BOOL;                // 计数器1完成标志
    bfin2 : BOOL;                // 保留
    istate : INT;                // 上电状态机
    icount : INT;                // 上电步骤计数
END_VAR

(*==============================================================================
  FB: Az_Ctrl_FB（方位轴 Azimuth 控制功能块）
  与 El_Ctrl_FB 结构完全相同，差异点:
    - 操作的 GVL 变量为 Az 系列（diAzTargetVel / bAzCtrlBitX / eAzErrorcode 等）
    - positionMode 加速度为 12 deg/s²（El 为 9 deg/s²）
    - positionMode 的 Kp=0.6（El 为 0.7），本控 programBootMode Kp=0.6
    - programBootMode 参数来自 PersistentVars.rAzXxx

  速度换算公式（通用）:
    diAzTargetVel [inc/s] = deg/s × 524288 / 360
==============================================================================*)

// =============================================================================
// 段 A: 轴停止或下电时清快速停止位 bit8
// =============================================================================
IF sStatus.Disabled OR(NOT sStatus.Moving)THEN
	bAzCtrlBit8 := FALSE;
END_IF

// =============================================================================
// 段 B: 全局错误复位
// =============================================================================
IF GVL.bError_Reset THEN
	sCtrl.iMode:=6;
	sLocal.iMode:=6;
	GVL.Error_code:=0;
END_IF
IF GVL.Error_code =0 THEN
	GVL.bError_Reset:=FALSE;
END_IF

// =============================================================================
// 段 C: CANopen 心跳超时（0x8130）自动恢复序列
// =============================================================================
IF GVL.eAzErrorcode = 16#8130 AND NOT tr THEN
	GVL.bAzCtrlBit7 := TRUE;
	tr:=TRUE;
	istate:=0;
	icount:=0;
	// 写入下电控制字
	GVL.bAzCtrlBit3 := FALSE;
	GVL.bAzCtrlBit0 := FALSE;
	GVL.bAzCtrlBit1 := FALSE;
	GVL.bAzCtrlBit2 := FALSE;
END_IF
IF tr THEN
	icount1 := icount1 + 1;
END_IF
IF icount1 > 101 THEN
	icount1 := 0;
	tr := FALSE;
	GVL.bAzCtrlBit7 := FALSE;
	bfin1 := TRUE;
END_IF
IF bfin1 THEN
	icount2 := icount2 + 1;
END_IF
IF icount2 > 101 THEN
	bfin1 := FALSE;
	icount2 := 0;
END_IF

// =============================================================================
// 段 D: 主控制逻辑
// =============================================================================
IF GVL.Error_code=0 AND GVL.eAzErrorcode = 0 AND NOT GVL.bAzCtrlBit7  AND NOT tr AND NOT bfin1 AND NOT bfin2 THEN

	// =========== 远控 ===========
	IF GVL.bLocalCtrl=FALSE THEN //远控
		IF sCtrl.iMode <> 1 THEN
			istate:=0;
			icount:=0;
		END_IF
		CASE sCtrl.iMode OF

			MODES.powerOff: // 下电
				IF NOT sStatus.Disabled THEN
					IF sStatus.Moving THEN // 运动中，先停止运动
						GVL.diAzTargetVel := 0;
						bAzCtrlBit8 := TRUE;
					ELSE
						// 写入下电控制字
						GVL.bAzCtrlBit3 := FALSE;
						GVL.bAzCtrlBit0 := FALSE;
						GVL.bAzCtrlBit1 := FALSE;
						GVL.bAzCtrlBit2 := FALSE;
					END_IF
				END_IF
				// 下电状态下持续调用 vpid1（保持内部状态稳定）
				vpid1(rKpbase:=1, rKibase:=0.01, rKpMax:=1, rKiMax:=0.01, rVelThreshold:=10,rTarget:=sCtrl.rPIDCmdPos,rFeedback:=rRealPos,rPosLimPositive:=sCtrl.rSoft_limit_Postive,
							rPosLimNegitive:=sCtrl.rSoft_limit_Negative,
								bPIDEnable:=sCtrl.bPIDEnable,rVelLim:=sCtrl.rVel_Limit,rKpScale:=0.02,rKiScale:=0.005,rElPos:=GVL.rFctPosReal_1-90,
								iThrehold:=sCtrl.rPIDThre,rPIDOutDir=>sCtrl.rPIDCmdVel);

			MODES.powerOn:  // 上电（DS402 三步序列）
				IF sStatus.Disabled THEN
					GVL.diAzTargetVel := 0;
					IF GVL.siAzMode <> 3 THEN // 上电时模式默认为3，速度模式
						GVL.siAzMode := 3;
					END_IF
					IF siAzMode = 3 THEN
						CASE istate OF
							0:
								GVL.bAzCtrlBit1 := TRUE;
								GVL.bAzCtrlBit2 := TRUE;
								icount := icount + 1;
								IF icount = 20 THEN
									icount:=0;
									istate:=1;
								END_IF
							1:
								GVL.bAzCtrlBit0 := TRUE;
								icount := icount + 1;
								IF icount = 20 THEN
									icount:=0;
									istate:=2;
								END_IF
							2:
								GVL.bAzCtrlBit3 := TRUE;
						END_CASE
					END_IF
				ELSE
					IF sStatus.Moving THEN
						GVL.diAzTargetVel := 0;
						bAzCtrlBit8 := TRUE;
					ELSE
						bAzCtrlBit8 := FALSE;
					END_IF
				END_IF

			MODES.positionMode: // 远控指向模式（加速度 12 deg/s²，Kp=0.6）
				IF NOT sStatus.Disabled THEN
					IF sCtrl.bStartAutoTrack THEN
						//自跟踪模式下，由误差电压直接驱动
						VelPID_1(rTarget:=sCtrl.rChanU + rRealPos,
								rFeedback:=rRealPos,
								rPosLimPositive:=sCtrl.rSoft_limit_Postive,
								rPosLimNegative:=sCtrl.rSoft_limit_Negative,
								rVelLim:=sCtrl.rVel_Limit,
								rKp:=1,//自跟踪PI系数3,0.02
								rKi:=0,
								rKd:=0,
								bPIDEnable:=sCtrl.bPIDEnable,
								iThreshold:= -1,
								rPIDOutput=>sCtrl.rPIDCmdVel);							
					ELSE
						//PID计算速度指令
						VelPID_1(rTarget:=sCtrl.rPosCmd,
							rFeedback:=rRealPos,
							rVelLim:=sCtrl.Pos_Vel,
							rPosLimPositive:=sCtrl.rSoft_limit_Postive,
							rPosLimNegative:=sCtrl.rSoft_limit_Negative,
							rKp:=0.6,//程引PI系数低带：1,0.002  高带：3,0.02
							rKi:=0,
							rKd:=0,
							bPIDEnable:=sCtrl.bPIDEnable,
							iThreshold:=sCtrl.rPIDThre,
							rPIDOutput=>sCtrl.rPIDCmdVel);
					END_IF
					GVL.diAzTargetVel := REAL_TO_DINT(sCtrl.rPIDCmdVel * 524288 / 360);
					GVL.diAzTargetAcc := REAL_TO_UDINT(12 * 524288 / 360);   //加速度 12 deg/s²
					GVL.diAzTargetDec := REAL_TO_UDINT(12 * 524288 / 360);   //减速度
				END_IF

			MODES.velocityMode://手控速度模式-远控模式
				IF NOT sStatus.Disabled THEN
					IF ABS(sCtrl.rVelCmd) <= sCtrl.rVel_Limit THEN
						GVL.diAzTargetVel := REAL_TO_DINT(sCtrl.rVelCmd * 524288 / 360);
					ELSIF sCtrl.rVelCmd > sCtrl.rVel_Limit THEN
						GVL.diAzTargetVel := REAL_TO_DINT(sCtrl.rVel_Limit * 524288 / 360);
					ELSE
						GVL.diAzTargetVel := REAL_TO_DINT(-sCtrl.rVel_Limit * 524288 / 360);
					END_IF
					GVL.diAzTargetAcc := REAL_TO_UDINT(sCtrl.rAcceleration * 524288 / 360);   //加速度
					GVL.diAzTargetDec := REAL_TO_UDINT(sCtrl.rDeceleration * 524288 / 360);   //减速度
				END_IF

			MODES.programBootMode://PID速度模式-正常模式 程引（变增益 vpid1）
				IF NOT sStatus.Disabled THEN
					IF sCtrl.bStartAutoTrack THEN
						// 程引+自跟踪
						vpid1(rKpbase:=Persistentvars.rAzKpBase, rKibase:=Persistentvars.rAzKiBase, rKpMax:=Persistentvars.rAzKpMax, rKiMax:=Persistentvars.rAzKiMax, rVelThreshold:=Persistentvars.rAzThre,rTarget:=sCtrl.rPIDCmdPos,rFeedback:=rRealPos,rPosLimPositive:=sCtrl.rSoft_limit_Postive,
							rPosLimNegitive:=sCtrl.rSoft_limit_Negative,
								bPIDEnable:=sCtrl.bPIDEnable,rVelLim:=sCtrl.rVel_Limit,rKpScale:=Persistentvars.rAzKpscale,rKiScale:=Persistentvars.rAzKiscale,rElPos:=GVL.rFctPosReal_1-90,
								iThrehold:=sCtrl.rPIDThre,rPIDOutDir=>sCtrl.rPIDCmdVel);							
					ELSE
						// 纯程引
						vpid1(rKpbase:=Persistentvars.rAzKpBase, rKibase:=Persistentvars.rAzKiBase, rKpMax:=Persistentvars.rAzKpMax, rKiMax:=Persistentvars.rAzKiMax, rVelThreshold:=Persistentvars.rAzThre,rTarget:=sCtrl.rPIDCmdPos,rFeedback:=rRealPos,rPosLimPositive:=sCtrl.rSoft_limit_Postive,
							rPosLimNegitive:=sCtrl.rSoft_limit_Negative,
								bPIDEnable:=sCtrl.bPIDEnable,rVelLim:=sCtrl.rVel_Limit,rKpScale:=Persistentvars.rAzKpscale,rKiScale:=Persistentvars.rAzKiscale,rElPos:=GVL.rFctPosReal_1-90,
								iThrehold:=sCtrl.rPIDThre,rPIDOutDir=>sCtrl.rPIDCmdVel);
						
					END_IF
					GVL.diAzTargetVel := REAL_TO_DINT(sCtrl.rPIDCmdVel * 524288 / 360);
					GVL.diAzTargetAcc := REAL_TO_UDINT(sCtrl.rAcceleration * 524288 / 360);   //加速度
					GVL.diAzTargetDec := REAL_TO_UDINT(sCtrl.rDeceleration * 524288 / 360);   //减速度
				END_IF

			MODES.reset://重置
				IF NOT sStatus.Disabled THEN
					IF sStatus.Moving THEN
						GVL.diAzTargetVel := 0;
						bAzCtrlBit8 := TRUE;
					ELSE
						bAzCtrlBit8 := FALSE;
					END_IF
				END_IF

			MODES.halt://待机
				IF NOT sStatus.Disabled THEN
					IF sStatus.Moving THEN
						GVL.diAzTargetVel := 0;
						bAzCtrlBit8 := TRUE;
					ELSE
						bAzCtrlBit8 := FALSE;
					END_IF
				END_IF
			
		END_CASE

	// =========== 本控 ===========
	ELSE // 本控
		IF sLocal.iMode <> 1 THEN
			istate:=0;
			icount:=0;
		END_IF
		CASE sLocal.iMode OF

			MODES.powerOff: // 下电
				IF NOT sStatus.Disabled THEN
					IF sStatus.Moving THEN // 运动中，先停止运动
						GVL.diAzTargetVel := 0;
						bAzCtrlBit8 := TRUE;
					ELSE
						// 写入下电控制字
						GVL.bAzCtrlBit3 := FALSE;
						GVL.bAzCtrlBit0 := FALSE;
						GVL.bAzCtrlBit1 := FALSE;
						GVL.bAzCtrlBit2 := FALSE;
					END_IF
				END_IF

			MODES.powerOn:  // 上电
				IF sStatus.Disabled THEN
					GVL.diAzTargetVel := 0;
					IF GVL.siAzMode <> 3 THEN // 上电时模式默认为3，速度模式
						GVL.siAzMode := 3;
					END_IF
					IF siAzMode = 3 THEN
						CASE istate OF
							0:
								GVL.bAzCtrlBit1 := TRUE;
								GVL.bAzCtrlBit2 := TRUE;
								icount := icount + 1;
								IF icount = 20 THEN
									icount:=0;
									istate:=1;
								END_IF
							1:
								GVL.bAzCtrlBit0 := TRUE;
								icount := icount + 1;
								IF icount = 20 THEN
									icount:=0;
									istate:=2;
								END_IF
							2:
								GVL.bAzCtrlBit3 := TRUE;
						END_CASE
					END_IF
				ELSE
					IF sStatus.Moving THEN
						GVL.diAzTargetVel := 0;
						bAzCtrlBit8 := TRUE;
					ELSE
						bAzCtrlBit8 := FALSE;
					END_IF
				END_IF

			MODES.velocityMode://手控速度模式-本控模式
				IF NOT sStatus.Disabled THEN
					IF ABS(sLocal.rVelCmd) <= sLocal.rVel_Limit THEN
						GVL.diAzTargetVel := REAL_TO_DINT(sLocal.rVelCmd * 524288 / 360);
					ELSIF sLocal.rVelCmd > sLocal.rVel_Limit THEN
						GVL.diAzTargetVel := REAL_TO_DINT(sLocal.rVel_Limit * 524288 / 360);
					ELSE
						GVL.diAzTargetVel := REAL_TO_DINT(-sLocal.rVel_Limit * 524288 / 360);
					END_IF
					GVL.diAzTargetAcc := REAL_TO_UDINT(sLocal.rAcceleration * 524288 / 360);   //加速度
					GVL.diAzTargetDec := REAL_TO_UDINT(sLocal.rDeceleration * 524288 / 360);   //减速度
				END_IF

			MODES.programBootMode://本控位置模式（普通 PID，Kp=0.6）
				IF NOT sStatus.Disabled THEN
					IF NOT sLocal.bPIDEnable THEN
						GVL.diAzTargetVel := 0;							
					ELSE
						IF NOT slocal.bStartAutoTrack THEN
							//PID计算速度指令
							 VelPID_2(rTarget:=sLocal.rPosCmd,
									 rFeedback:=rRealPos,
									 rPosLimPositive:=sLocal.rSoft_limit_Postive,//软限位
									 rPosLimNegative:=sLocal.rSoft_limit_Negative,
									 rKp:=0.6,
									 rKi:=0,
									 rKd:=0,
									 iThreshold:=sLocal.rPIDThre,
									 bPIDEnable:=sLocal.bPIDEnable,
									 rVelLim:=sLocal.Pos_Vel,
									 rPIDOutput=>sLocal.rPIDCmdVel);//普通PID
						ELSE
							//PID计算速度指令
							 VelPID_2(rTarget:=sLocal.rChanU + rRealPos,
								rFeedback:=rRealPos,
								rPosLimPositive:=sLocal.rSoft_limit_Postive,
								rPosLimNegative:=sLocal.rSoft_limit_Negative,
								rVelLim:=sLocal.rVel_Limit,
								rKp:=1,//自跟踪PI系数3,0.02
								rKi:=0,
								rKd:=0,
								bPIDEnable:=sLocal.bPIDEnable,
								iThreshold:= -1,
								rPIDOutput=>sLocal.rPIDCmdVel);//普通PID
						END_IF
						
					END_IF
					GVL.diAzTargetVel := REAL_TO_DINT(sLocal.rPIDCmdVel * 524288 / 360);
					GVL.diAzTargetAcc := REAL_TO_UDINT(12 * 524288 / 360);   //加速度
					GVL.diAzTargetDec := REAL_TO_UDINT(12 * 524288 / 360);   //减速度
				END_IF

			MODES.reset://重置
			// 是否需要
			MODES.halt://待机
				IF NOT sStatus.Disabled THEN
					IF sStatus.Moving THEN
						GVL.diAzTargetVel := 0;
						bAzCtrlBit8 := TRUE;
					ELSE
						bAzCtrlBit8 := FALSE;
					END_IF
				END_IF
			
		END_CASE
	END_IF

// =============================================================================
// 段 E: 全局错误时强制停轴，超时后强制下电
// =============================================================================
ELSIF GVL.Error_code<>0 AND GVL.eAzErrorcode = 0 AND NOT GVL.bAzCtrlBit7  AND NOT tr AND NOT bfin1 AND NOT bfin2 THEN
	// 出现错误，轴停止运动
	GVL.diAzTargetVel := 0;
	bAzCtrlBit8 := TRUE;
	TON_0(IN:=bAzCtrlBit8,PT:=T#1S,Q=>,ET=>);//判断stop0执行是否超时,若超时强制下电（手动复位）
	IF TON_0.Q THEN
		bTick:=TRUE;
	END_IF
	IF bTick AND sStatus.Moving THEN // 超时强制下电
		// 写入下电控制字
		GVL.bAzCtrlBit3 := FALSE;
		GVL.bAzCtrlBit0 := FALSE;
		GVL.bAzCtrlBit1 := FALSE;
		GVL.bAzCtrlBit2 := FALSE;
	END_IF
END_IF

END_FUNCTION_BLOCK

// Device/Application/Ti_Ctrl_FB
FUNCTION_BLOCK Ti_Ctrl_FB

VAR_INPUT
    sLocal : AxisCrtlStruct;     // 本控命令结构体
    sCtrl : AxisCrtlStruct;      // 远控命令结构体
    sStatus : AxisStatus;        // 轴状态
    sVisible : AxisVisible;      // HMI 可视化（此 FB 未直接使用）
    rRealPos : REAL;             // 编码器实际位置 (deg)
    rPosLimK : REAL;             // 备用限位系数
END_VAR

VAR_OUTPUT
    logicError : INT;            // 保留
END_VAR

VAR
    VelPID_1 : PID;              // positionMode / programBootMode 远控用
    VelPID_2 : PID;              // 本控 programBootMode 用
    TON_0 : TON;                 // 超时 1s 强制下电计时器
    bTick : BOOL;                // stop0 超时标志
    tr : BOOL;                   // 心跳恢复进行中标志
    icount1 : INT;               // 心跳恢复计数器1
    icount2 : INT;               // 心跳恢复计数器2
    icount3 : INT;               // 备用
    bfin1 : BOOL;                // 计数器1完成标志
    bfin2 : BOOL;                // 保留
    istate : INT;                // 上电状态机
    icount : INT;                // 上电步骤计数
END_VAR

(*==============================================================================
  FB: Ti_Ctrl_FB（倾斜轴 Tilt 控制功能块）
  与 El_Ctrl_FB / Az_Ctrl_FB 结构基本相同，主要差异:
    - 操作的 GVL 变量为 Ti 系列（diTiTargetVel / bTiCtrlBitX / eTiErrorcode 等）
    - 无 vpid1（Ti 轴不做变增益，programBootMode 远控直接用 VelPID_1）
    - positionMode 加速度为 10 deg/s²
    - positionMode bStartAutoTrack 分支注释掉（Ti 无自跟踪需求）
    - programBootMode 本控用 VelPID_2，参数直接来自 sLocal.rP/rI/rD
    - programBootMode 远控 bStartAutoTrack=TRUE 时调用 VelPID_1（非 vpid1）

  速度换算公式（通用）:
    diTiTargetVel [inc/s] = deg/s × 524288 / 360
==============================================================================*)

// =============================================================================
// 段 A: 轴停止或下电时清快速停止位 bit8
// =============================================================================
IF sStatus.Disabled OR(NOT sStatus.Moving)THEN
	bTiCtrlBit8 := FALSE;
END_IF

// =============================================================================
// 段 B: 全局错误复位
// =============================================================================
IF GVL.bError_Reset THEN
	sCtrl.iMode:=6;
	sLocal.iMode:=6;
	GVL.Error_code:=0;
END_IF
IF GVL.Error_code =0 THEN
	GVL.bError_Reset:=FALSE;
END_IF

// =============================================================================
// 段 C: CANopen 心跳超时（0x8130）自动恢复序列
// =============================================================================
IF GVL.eTiErrorcode = 16#8130 AND NOT tr THEN
	GVL.bTiCtrlBit7 := TRUE;
	tr:=TRUE;
	istate:=0;
	icount:=0;
	// 写入下电控制字
	GVL.bTiCtrlBit3 := FALSE;
	GVL.bTiCtrlBit0 := FALSE;
	GVL.bTiCtrlBit1 := FALSE;
	GVL.bTiCtrlBit2 := FALSE;
END_IF
IF tr THEN
	icount1 := icount1 + 1;
END_IF
IF icount1 > 101 THEN
	icount1 := 0;
	tr := FALSE;
	GVL.bTiCtrlBit7 := FALSE;
	bfin1 := TRUE;
END_IF
IF bfin1 THEN
	icount2 := icount2 + 1;
END_IF
IF icount2 > 101 THEN
	bfin1 := FALSE;
	icount2 := 0;
END_IF

// =============================================================================
// 段 D: 主控制逻辑
// =============================================================================
IF GVL.Error_code=0 AND GVL.eTiErrorcode = 0 AND NOT GVL.bTiCtrlBit7  AND NOT tr AND NOT bfin1 AND NOT bfin2 THEN

	// =========== 远控 ===========
	IF GVL.bLocalCtrl=FALSE THEN //远控
		IF sCtrl.iMode <> 1 THEN
			istate:=0;
			icount:=0;
		END_IF
		CASE sCtrl.iMode OF

			MODES.powerOff: // 下电
				IF NOT sStatus.Disabled THEN
					IF sStatus.Moving THEN // 运动中，先停止运动
						GVL.diTiTargetVel := 0;
						bTiCtrlBit8 := TRUE;
					ELSE
						// 写入下电控制字
						GVL.bTiCtrlBit3 := FALSE;
						GVL.bTiCtrlBit0 := FALSE;
						GVL.bTiCtrlBit1 := FALSE;
						GVL.bTiCtrlBit2 := FALSE;
					END_IF
				END_IF

			MODES.powerOn:  // 上电（DS402 三步序列）
				IF sStatus.Disabled THEN
					GVL.diTiTargetVel := 0;
					IF GVL.siTiMode <> 3 THEN // 上电时模式默认为3，速度模式
						GVL.siTiMode := 3;
					END_IF
					IF siTiMode = 3 THEN
						CASE istate OF
							0:
								GVL.bTiCtrlBit1 := TRUE;
								GVL.bTiCtrlBit2 := TRUE;
								icount := icount + 1;
								IF icount = 20 THEN
									icount:=0;
									istate:=1;
								END_IF
							1:
								GVL.bTiCtrlBit0 := TRUE;
								icount := icount + 1;
								IF icount = 20 THEN
									icount:=0;
									istate:=2;
								END_IF
							2:
								GVL.bTiCtrlBit3 := TRUE;
						END_CASE
					END_IF
				ELSE
					IF sStatus.Moving THEN
						GVL.diTiTargetVel := 0;
						bTiCtrlBit8 := TRUE;
					ELSE
						bTiCtrlBit8 := FALSE;
					END_IF
				END_IF

			MODES.positionMode: // 远控指向模式（加速度 10 deg/s²，Kp=0.8）
				IF NOT sStatus.Disabled THEN
					IF sCtrl.bStartAutoTrack THEN
						// Ti 轴自跟踪分支已注释掉，实际走 ELSE
						(*
						VelPID_1(rTarget:=sCtrl.rChanU + rRealPos,
								rFeedback:=rRealPos,
								rPosLimPositive:=sCtrl.rSoft_limit_Postive,
								rPosLimNegative:=sCtrl.rSoft_limit_Negative,
								rVelLim:=sCtrl.rVel_Limit,
								rKp:=sCtrl.rP_AutoTrack,//自跟踪PI系数3,0.02
								rKi:=sCtrl.rI_AutoTrack,
								rKd:=sCtrl.rD,
								bPIDEnable:=sCtrl.bPIDEnable,
								iThreshold:= -1,
								rPIDOutput=>sCtrl.rPIDCmdVel);
*)							
					ELSE
						//PID计算速度指令
						VelPID_1(rTarget:=sCtrl.rPosCmd,
							rFeedback:=rRealPos,
							rVelLim:=sCtrl.Pos_Vel,
							rPosLimPositive:=sCtrl.rSoft_limit_Postive,
							rPosLimNegative:=sCtrl.rSoft_limit_Negative,
							rKp:=0.8,//程引PI系数地带：1,0.002  高带：3,0.02
							rKi:=0,
							rKd:=0,
							bPIDEnable:=sCtrl.bPIDEnable,
							iThreshold:=sCtrl.rPIDThre,
							rPIDOutput=>sCtrl.rPIDCmdVel);
					END_IF
					GVL.diTiTargetVel := REAL_TO_DINT(sCtrl.rPIDCmdVel * 524288 / 360);
					GVL.diTiTargetAcc := REAL_TO_UDINT(10 * 524288 / 360);   //加速度 10 deg/s²
					GVL.diTiTargetDec := REAL_TO_UDINT(10 * 524288 / 360);   //减速度
				END_IF

			MODES.velocityMode://手控速度模式-远控模式
				IF NOT sStatus.Disabled THEN
					IF ABS(sCtrl.rVelCmd) <= sCtrl.rVel_Limit THEN
						GVL.diTiTargetVel := REAL_TO_DINT(sCtrl.rVelCmd * 524288 / 360);
					ELSIF sCtrl.rVelCmd > sCtrl.rVel_Limit THEN
						GVL.diTiTargetVel := REAL_TO_DINT(sCtrl.rVel_Limit * 524288 / 360);
					ELSE
						GVL.diTiTargetVel := REAL_TO_DINT(-sCtrl.rVel_Limit * 524288 / 360);
					END_IF
					GVL.diTiTargetAcc := REAL_TO_UDINT(sCtrl.rAcceleration * 524288 / 360);   //加速度
					GVL.diTiTargetDec := REAL_TO_UDINT(sCtrl.rDeceleration * 524288 / 360);   //减速度
				END_IF

			MODES.programBootMode://PID速度模式-正常模式 程引（Ti 轴用 VelPID_1，非 vpid）
				IF NOT sStatus.Disabled THEN
					IF sCtrl.bStartAutoTrack THEN
						// 程引+自跟踪：误差电压叠加到插值位置
						VelPID_1(rTarget:=sCtrl.rChanU + rRealPos,
								rFeedback:=rRealPos,
								rPosLimPositive:=sCtrl.rSoft_limit_Postive,
								rPosLimNegative:=sCtrl.rSoft_limit_Negative,
								rVelLim:=sCtrl.rVel_Limit,
								rKp:=sCtrl.rP_AutoTrack,//自跟踪PI系数3,0.02
								rKi:=sCtrl.rI_AutoTrack,
								rKd:=sCtrl.rD,
								bPIDEnable:=sCtrl.bPIDEnable,
								iThreshold:= -1,
								rPIDOutput=>sCtrl.rPIDCmdVel);							
					ELSE
						//PID计算速度指令（参数来自 sCtrl.rP/rI/rD，由 Modbus/上位机配置）
						VelPID_1(rTarget:=sCtrl.rPIDCmdPos,
							rFeedback:=rRealPos,
							rVelLim:=sCtrl.rVel_Limit,
							rPosLimPositive:=sCtrl.rSoft_limit_Postive,
							rPosLimNegative:=sCtrl.rSoft_limit_Negative,
							rKp:=sCtrl.rP,//程引PI系数地带：1,0.002  高带：3,0.02
							rKi:=sCtrl.rI,
							rKd:=sCtrl.rD,
							bPIDEnable:=sCtrl.bPIDEnable,
							iThreshold:=sCtrl.rPIDThre,
							rPIDOutput=>sCtrl.rPIDCmdVel);
					END_IF
					GVL.diTiTargetVel := REAL_TO_DINT(sCtrl.rPIDCmdVel * 524288 / 360);
					GVL.diTiTargetAcc := REAL_TO_UDINT(sCtrl.rAcceleration * 524288 / 360);   //加速度
					GVL.diTiTargetDec := REAL_TO_UDINT(sCtrl.rDeceleration * 524288 / 360);   //减速度
				END_IF

			MODES.reset://重置
				IF NOT sStatus.Disabled THEN
					IF sStatus.Moving THEN
						GVL.diTiTargetVel := 0;
						bTiCtrlBit8 := TRUE;
					ELSE
						bTiCtrlBit8 := FALSE;
					END_IF
				END_IF

			MODES.halt://待机
				IF NOT sStatus.Disabled THEN
					IF sStatus.Moving THEN
						GVL.diTiTargetVel := 0;
						bTiCtrlBit8 := TRUE;
					ELSE
						bTiCtrlBit8 := FALSE;
					END_IF
				END_IF
			
		END_CASE

	// =========== 本控 ===========
	ELSE // 本控
		IF sLocal.iMode <> 1 THEN
			istate:=0;
			icount:=0;
		END_IF
		CASE sLocal.iMode OF

			MODES.powerOff: // 下电
				IF NOT sStatus.Disabled THEN
					IF sStatus.Moving THEN // 运动中，先停止运动
						GVL.diTiTargetVel := 0;
						bTiCtrlBit8 := TRUE;
					ELSE
						// 写入下电控制字
						GVL.bTiCtrlBit3 := FALSE;
						GVL.bTiCtrlBit0 := FALSE;
						GVL.bTiCtrlBit1 := FALSE;
						GVL.bTiCtrlBit2 := FALSE;
					END_IF
				END_IF

			MODES.powerOn:  // 上电
				IF sStatus.Disabled THEN
					GVL.diTiTargetVel := 0;
					IF GVL.siTiMode <> 3 THEN // 上电时模式默认为3，速度模式
						GVL.siTiMode := 3;
					END_IF
					IF siTiMode = 3 THEN
						CASE istate OF
							0:
								GVL.bTiCtrlBit1 := TRUE;
								GVL.bTiCtrlBit2 := TRUE;
								icount := icount + 1;
								IF icount = 20 THEN
									icount:=0;
									istate:=1;
								END_IF
							1:
								GVL.bTiCtrlBit0 := TRUE;
								icount := icount + 1;
								IF icount = 20 THEN
									icount:=0;
									istate:=2;
								END_IF
							2:
								GVL.bTiCtrlBit3 := TRUE;
						END_CASE
					END_IF
				ELSE
					IF sStatus.Moving THEN
						GVL.diTiTargetVel := 0;
						bTiCtrlBit8 := TRUE;
					ELSE
						bTiCtrlBit8 := FALSE;
					END_IF
				END_IF

			MODES.velocityMode://手控速度模式-本控模式
				IF NOT sStatus.Disabled THEN
					IF ABS(sLocal.rVelCmd) <= sLocal.rVel_Limit THEN
						GVL.diTiTargetVel := REAL_TO_DINT(sLocal.rVelCmd * 524288 / 360);
					ELSIF sLocal.rVelCmd > sLocal.rVel_Limit THEN
						GVL.diTiTargetVel := REAL_TO_DINT(sLocal.rVel_Limit * 524288 / 360);
					ELSE
						GVL.diTiTargetVel := REAL_TO_DINT(-sLocal.rVel_Limit * 524288 / 360);
					END_IF
					GVL.diTiTargetAcc := REAL_TO_UDINT(sLocal.rAcceleration * 524288 / 360);   //加速度
					GVL.diTiTargetDec := REAL_TO_UDINT(sLocal.rDeceleration * 524288 / 360);   //减速度
				END_IF

			MODES.programBootMode://本控位置模式（普通 PID，参数来自 sLocal.rP/rI/rD）
				IF NOT sStatus.Disabled THEN
					IF NOT sLocal.bPIDEnable THEN
						GVL.diTiTargetVel := 0;							
					ELSE
						//PID计算速度指令
						 VelPID_2(rTarget:=sLocal.rPosCmd,
							     rFeedback:=rRealPos,
								 rPosLimPositive:=sLocal.rSoft_limit_Postive,//软限位
								 rPosLimNegative:=sLocal.rSoft_limit_Negative,
								 rKp:=sLocal.rP,
								 rKi:=sLocal.rI,
								 rKd:=sLocal.rD,
								 iThreshold:=sLocal.rPIDThre,
								 bPIDEnable:=sLocal.bPIDEnable,
								 rVelLim:=sLocal.Pos_Vel,
								 rPIDOutput=>sLocal.rPIDCmdVel);//普通PID
					END_IF
					GVL.diTiTargetVel := REAL_TO_DINT(sLocal.rPIDCmdVel * 524288 / 360);
					GVL.diTiTargetAcc := REAL_TO_UDINT(sLocal.rAcceleration * 524288 / 360);   //加速度
					GVL.diTiTargetDec := REAL_TO_UDINT(sLocal.rDeceleration * 524288 / 360);   //减速度
				END_IF

			MODES.reset://重置
			// 是否需要
			MODES.halt://待机
				IF NOT sStatus.Disabled THEN
					IF sStatus.Moving THEN
						GVL.diTiTargetVel := 0;
						bTiCtrlBit8 := TRUE;
					ELSE
						bTiCtrlBit8 := FALSE;
					END_IF
				END_IF
			
		END_CASE
	END_IF

// =============================================================================
// 段 E: 全局错误时强制停轴，超时后强制下电
// =============================================================================
ELSIF GVL.Error_code<>0 AND GVL.eTiErrorcode = 0 AND NOT GVL.bTiCtrlBit7  AND NOT tr AND NOT bfin1 AND NOT bfin2 THEN
	// 出现错误，轴停止运动
	GVL.diTiTargetVel := 0;
	bTiCtrlBit8 := TRUE;
	TON_0(IN:=bTiCtrlBit8,PT:=T#1S,Q=>,ET=>);//判断stop0执行是否超时,若超时强制下电（手动复位）
	IF TON_0.Q THEN
		bTick:=TRUE;
	END_IF
	IF bTick AND sStatus.Moving THEN // 超时强制下电
		// 写入下电控制字
		GVL.bTiCtrlBit3 := FALSE;
		GVL.bTiCtrlBit0 := FALSE;
		GVL.bTiCtrlBit1 := FALSE;
		GVL.bTiCtrlBit2 := FALSE;
	END_IF
END_IF

END_FUNCTION_BLOCK

// Device/Application/AutoTrackingCal
PROGRAM AutoTrackingCal

VAR
    rChanUa : REAL;                    // 处理后方位误差 (V)，→ Az 自跟踪
    rChanUe : REAL;                    // 处理后俯仰误差 (V)，→ El 自跟踪
    rChanAGC : REAL;                   // 当前通道 AGC
    bChanLock : BOOL;                  // 通道锁定（保留）
    iCountATLock : INT;
    iState : INT;                      // 跟踪通道选择：1=通道1, 2=通道2
    rAzSum : LREAL;                    // 方位累积拉偏
    rElSum : LREAL;                    // 俯仰累积拉偏
    rDirSenFac : REAL;                 // 方向灵敏度系数（除数）
    rCurentEl : LREAL;                 // 当前俯仰角弧度 (rFctPosReal_1-90)
    rk : LREAL;                        // 累积增益（用于 rAzSum/rElSum）
    rChanUaLocal : REAL;               // 本控方位误差（未见赋值逻辑）
    rChanUeLocal : REAL;               // 本控俯仰误差（未见赋值逻辑）
END_VAR



(*==============================================================================
  PRG: AutoTrackingCal（自跟踪误差电压处理）
  任务: Canopen 10ms
  输入: GVL.Chan1Ua/Ue/AGC/Lock（由 READ_485 写入）
  输出（程序内变量，供 *_ctrl_1 引用）:
    rChanUa  — 方位误差电压（已÷灵敏度、÷cos(俯仰)）
    rChanUe  — 俯仰误差电压（已÷灵敏度）
    rAzSum / rElSum — 累积拉偏量（当前未回写到 GVL）
  使用:
    El_ctrl_1: rChanUe → rChanU / rAuToStepBias
    Az_ctrl_1: -rChanUa → rChanU / rAuToStepBias
  注意:
    rDirSenFac、rk 在导出代码中未见赋值，可能来自 Modbus/HMI 或需人工确认
    rChanUaLocal / rChanUeLocal 未见赋值，本控自跟踪可能依赖未初始化值（原工程保留）
==============================================================================*)
(* 旧版按 iState 直接映射 GVL 通道，已注释 *)

//iState:=modbusSlave.Trace_Num;//跟踪支路选择
iState:=1;                             // 固定使用跟踪接收机 1

CASE iState OF 
	1://使用跟踪接收机1 且锁定标识为True
		// ----- 自跟踪使能且（锁定或 SecurityCheck 误差电压足够小）-----
		IF GVL.bStartTrack AND (GVL.Chan1Lock OR Securitycheck.bErrorLock) THEN
			// 方位：原始 Ua → ÷灵敏度 → ÷cos(El) 补偿大仰角时方位耦合
			rChanUa:=GVL.Chan1Ua;
			rChanUa:=rChanUa/rDirSenFac;
			rCurentEl:=(rFctPosReal_1-90)*3.1415926535897/180.0;
			rChanUa:=rChanUa/COS(rCurentEl);
			
			// 俯仰：原始 Ue → ÷灵敏度
			rChanUe:=GVL.Chan1Ue;
			rChanUe:=rChanUe/rDirSenFac;
			rChanAGC:=GVL.Chan1AGC;
			
			// 累积量（供扩展；当前 *_ctrl_1 主要用瞬时 rChanUa/Ue）
			rAzSum:=rAzSum+rk*rChanUa/1000.0;
			rElSum:=rElSum+rk*rChanUe/1000.0;
		ELSE
			rAzSum:=0;
			rElSum:=0;
			rChanUa:=0;
			rChanUe:=0;
		END_IF
		
	2://使用跟踪接收机2 且锁定标识为True
		rChanUa:=GVL.Chan2Ua;
		rChanUe:=GVL.Chan2Ue;
		rChanAGC:=GVL.Chan2AGC;
		
	3://锁定标识符为False
		//bChanLock:=FALSE;
END_CASE

END_PROGRAM

// Device/Application/READ_485
PROGRAM READ_485
VAR
    com_init : gcan.FB_Com_Init;
    com_read : gcan.FB_Com_Read;
    com_write : gcan.FB_Com_Write;
    m_uiError : UINT;
    m_out : BOOL;
    isFirst : BOOL;
    mPort : BYTE;                      // 2 = 485 口
    recSize : UINT;
    recBuf : ARRAY[0..19] OF BYTE;     // 原始接收缓冲（对外可读 recBuf[1] 等）
    recData : ARRAY[0..8] OF BYTE;     // 旧协议 0x7E 帧解析用（已注释）
    wAGC : WORD;
    iUa : INT;
    iUe : INT;
    iChan1DataLen : UINT;
    chan1_i : INT;
    chan1_j : INT;
    Word2Bit1 : Word2Bit;              // AGC 高低字节 → WORD
    Word2Bit2 : Word2Bit;              // Ua → INT
    Word2Bit3 : Word2Bit;              // Ue → INT
    rUagcTemp : REAL;
    rUaTemp : REAL;
    rUeTemp : REAL;
    btest : BOOL;
    btest2 : BOOL;
    rSData : REAL;                     // 信号分量（DWORD 差）
    rQData : REAL;                     // 噪声分量
    Dword2Bit1 : Dword2Bit;            // recBuf[8..11] → DWORD
    Dword2Bit2 : Dword2Bit;            // recBuf[12..15] → DWORD
    Chan1EB_N0 : REAL;                 // 等效 Eb/N0 (dB)，SecurityCheck.bLockSearch 用
    bEBN0Lock : BOOL;                  // 信噪比锁定标志（与模式/失锁计数相关）
    icount0 : INT;                     // recBuf[1]=0 累计，>400 清 bEBN0Lock
END_VAR



(*==============================================================================
  PRG: READ_485（跟踪接收机 RS485 通信）
  任务: SerialCom 5ms（与 GPRMC_1 同任务，端口不同）
  硬件: GCAN 串口 mPort=2（485），19200 8N1
  作用:
    - 读跟踪接收机上报帧 → 解析 AGC、Ua、Ue、锁定、Eb/N0
    - 写入 GVL.Chan1AGC / Chan1Ua / Chan1Ue / Chan1Lock
    - 输出 Chan1EB_N0、recBuf[1]、bEBN0Lock 供 SecurityCheck / 捕获扫描
  帧布局（当前简化协议，非 0x7E 定界）:
    recBuf[1]     — 锁定标志 (1=锁定)
    recBuf[2..3]  — AGC 原始 WORD
    recBuf[4..5]  — 方位误差 Ua 原始 INT
    recBuf[6..7]  — 俯仰误差 Ue 原始 INT
    recBuf[8..15] — Eb/N0 用两路 DWORD 算信噪比
==============================================================================*)

mPort:=2;								//串口端口号设定

// ----- 首次上电：485 初始化 19200 -----
IF isFirst THEN
	com_init(
	EN_IN:=TRUE,
	xEnable:=TRUE,
	bPort:=mPort,
	uiBaudrate:=19200,
	bParity:=0,
	bDatabits:=8,
	bStopbits:=1,
	EN_OUT=>m_out,
	uiError=>m_uiError);
	isfirst:=FALSE;

ELSE
	com_read(
	EN_in:=TRUE,
	bPort:=mPort,
	p_brxdata:=ADR(recBuf),
	uiMaxsize:=20,
	EN_out=>m_out,
	uiRecSize=>recSize,
	uierror=>m_uierror);
	
	// ----- 段 1: 锁定标志 → GVL.Chan1Lock -----
	//GVL.Chan1Lock := BYTE_TO_BOOL(recBuf[1]);
	IF recBuf[1] = 1 AND GVL.Chan1AGC >= GVL.Chanthreshold THEN
		GVL.Chan1Lock := TRUE;
	ELSE
		GVL.Chan1Lock := FALSE;
	END_IF

	// ----- 段 2: 按字节拼接 WORD/INT（Word2Bit UNION）-----
	Word2Bit1.Apart_Byte[1] := recBuf[2];
	Word2Bit1.Apart_Byte[2] := recBuf[3];
	wAGC:=Word2Bit1.Apart_Word;
	
	Word2Bit2.Apart_Byte[1] := recBuf[4];
	Word2Bit2.Apart_Byte[2] := recBuf[5];
	iUa:=Word2Bit2.Apart_INT;
	
	Word2Bit3.Apart_Byte[1] := recBuf[6];
	Word2Bit3.Apart_Byte[2] := recBuf[7];
	iUe:=Word2Bit3.Apart_INT;

	// ----- 段 3: 换算为物理量并限幅后写 GVL -----
	// Ua/Ue: ±5V 满量程对应 INT±2048；AGC: 5 - (raw×5/76) 越大信号越强
	IF ABS(INT_TO_REAL(iUa) * 5 / 2048) <= 5 AND ABS(INT_TO_REAL(iUe) * 5 / 2048) <= 5 AND ABS((WORD_TO_REAL(wAGC) * 5 / 76)) <=5 THEN
		GVL.Chan1Ua := INT_TO_REAL(iUa) * 5 / 2048;
		GVL.Chan1Ue := INT_TO_REAL(iUe) * 5 / 2048;
		GVL.Chan1AGC := 5 - (WORD_TO_REAL(wAGC) * 5 / 76);
	END_IF
	
	// ----- 段 4: Eb/N0 估算（两 DWORD，字节序见 Dword2Bit 填入顺序）-----
	Dword2Bit1.Apart_Byte[3] := recBuf[8];
	Dword2Bit1.Apart_Byte[4] := recBuf[9];
	Dword2Bit1.Apart_Byte[1] := recBuf[10];
	Dword2Bit1.Apart_Byte[2] := recBuf[11];	
	
	Dword2Bit2.Apart_Byte[3] := recBuf[12];
	Dword2Bit2.Apart_Byte[4] := recBuf[13];
	Dword2Bit2.Apart_Byte[1] := recBuf[14];
	Dword2Bit2.Apart_Byte[2] := recBuf[15];	
	
	rQData:=DWORD_TO_REAL(Dword2Bit2.Apart_DWORD);
	rSData:=DWORD_TO_REAL(Dword2Bit1.Apart_DWORD)-rQData;
	
	IF rSData<>0  AND rQData<>0  THEN
		Chan1EB_N0 := 10*LOG(ABS(rSData/rQData))+3.8;
	ELSE
		Chan1EB_N0 := 0;
	END_IF
	
	// ----- 段 5: bEBN0Lock — 程引/指向且 Eb/N0≥29 或 ACU 请求自跟踪 -----
	IF ((GVL.Axis1Remote.iMode = 2 OR GVL.Axis1Remote.iMode = 4) AND Chan1EB_N0 >= 29)AND READ_485.recBuf[1] = 1 OR Modbus_Slave.bStartTrackAcu THEN
		icount0:=0;
		bEBN0Lock := TRUE;
	END_IF
	// 锁定字节为 0 时累计；超 400 拍或下电则清 bEBN0Lock
	IF ( GVL.Axis1Remote.iMode = 4 or GVL.Axis1Remote.iMode =2 ) AND recBuf[1] = 0 THEN
		icount0:=icount0+1;
	END_IF
	IF icount0 > 400 OR (GVL.Axis1Remote.iMode = 0 OR GVL.Axis1Remote.iMode = 0) THEN
		icount0 := 401;
		bEBN0Lock := FALSE;
	END_IF
END_IF

(* 旧版 0x7E 定界帧解析整段已注释 *)

END_PROGRAM

// Device/Application/扫描搜索/AGCMaxSearch_PB_1
FUNCTION_BLOCK AGCMaxSearch_PB_1 //双轴静止星步进跟踪使用的代码
VAR_INPUT
	bstart:BOOL;//模块开始标识
	rAGCNow:REAL;//当前AGC值
	btrig:BOOL;//触发一次
	rStepBiasNow:REAL;//当前拉偏量 //用来判断此次搜索是否有效
	bAutoTracking:BOOL;// 自跟踪标识
	bStop:BOOL;//满足ua ue很小
	
	rCurrentPos:REAL;//当前位置
	rInterPos:REAL;//插值位置
	//rOutStepBias:REAL;//外部拉偏量
END_VAR
VAR_OUTPUT
	
	rAGCMaxBias:REAL;//输出AGC最强时的拉偏量 单位为°
	bSucess :BOOL;//数出模块是否成功
	rStepBias:REAL;//步进量
END_VAR
VAR
	ton:Standard.TON;
	rTrg:Standard.R_TRIG;//初始化上升沿检测器
	rAGCInit:REAL:=0;//初始化AGC
	rPrevAGC:REAL:=0;//上一步的AGC值 单位为V
	rBiasInit:REAL;//初始化拉偏量
	
	iCountStep:INT:=0;//计步数
	toN1: Standard.Ton;//计时器 定时触发上升沿 
	
	rDirection: INT:=1;
	rSearchNextStepTarget:REAL;//搜索当前目标位置 单位为°
	rStep:REAL:=0.0003;//步进值
	rSensitivity:REAL:=0.05;//反向灵敏度
	iCountStopMax:INT:=20;//停止计数上限
	
	rLastDirection:INT;//上一次方向，判断是否换向
	iCountDirChange:INT;//换向标识
	rAGCMaxPos:REAL;//信号最强位置
	
	rAGCLastrecord: REAL;
	iStatus: INT;
	iCountStop1:INT;//第一阶段停止标识 (正向)
	iCountStop2:INT;//(反向)
	
	rAGCMaxValue: REAL;//AGC最大值
	
	//新加的
	iCountSearchRight:INT;//搜索方向正确，提前结束标识
	
	bSearchRight:BOOL;//搜索正确标识
	//模块指行完成标识
	iCountBlockEnd:INT;//用来计数确认已达到最强位置
	iCountBlockEndMax:INT:=500;//到位计数上限
END_VAR


(*==============================================================================
  FB: AGCMaxSearch_PB_1（AGC 峰值搜索：单轴拉偏搜索）
  调用者: `Az_ctrl_1` / `El_ctrl_1`
  目标: 在指向(mode2)或程引(mode4)时，沿单轴正/负方向试探移动 rStepBias，
        找到使 AGC 最大的位置偏置 rAGCMaxBias，并在到位稳定后置 bSucess

  关键变量含义:
    rStepBias      — 当前偏置输出（逐步累加 rDirection*rStep）
    rAGCMaxBias    — 历史最大 AGC 对应的偏置
    rAGCInit       — 启动时 AGC 基线
    rSensitivity   — 判定“AGC 明显下降/上升”的阈值，用于决定停止/换向
    iCountDirChange— 换向次数；=2 后进入“回到峰值位置并等待稳定”阶段

  完成判定:
    - 偏置回到 rAGCMaxBias 后，(rInterPos+rStepBias) 与 rCurrentPos 误差持续小于 0.002
    - 持续计数超过 iCountBlockEndMax 后，再用 TON(1s) 确认稳定 → bSucess=TRUE
==============================================================================*)

rTrg(CLK:=bstart,Q=>);

IF rTrg.Q THEN
	rAGCInit:=rAGCNow;
	rAGCMaxValue:=rAGCNow;
	//rBiasInit:=rCurrentPos-rInterPos;//获取启动时的拉偏量
END_IF

IF bstart THEN
	//搜索换向两次
	IF iCountDirChange=2 THEN
		rSearchNextStepTarget:=rAGCMaxBias;
		IF rStepBias< rSearchNextStepTarget THEN 
			rStepBias:=rStepBias+rStep;
		ELSIF rStepBias> rSearchNextStepTarget THEN
			rStepBias:=rStepBias-rStep;
		ELSE
			rStepBias:=rStepBias;
		END_IF
		
		IF ABS((rInterPos+rStepBias)-rCurrentPos)<0.002 THEN //若位置达到最强位置，则输出成功 //可能只是路过这里,需要持续
			//需要判断稳定
			iCountBlockEnd:=iCountBlockEnd+1;
		ELSE
			iCountBlockEnd:=0;
		END_IF
		IF iCountBlockEnd>iCountBlockEndMax THEN
			iCountBlockEnd:=iCountBlockEndMax+1;
			//用TON1秒后触发
			ton(IN:=TRUE,PT:=T#1S,Q=>,ET=>);
		END_IF
		IF ton.Q THEN
			bSucess:=TRUE;
		END_IF
	ELSE
		rStepBias:=rStepBias+rDirection*rStep;
		IF rDirection<0 THEN
			//若是向小走
			IF rCurrentPos<rInterPos THEN
				IF rAGCNow<rAGCMaxValue-rSensitivity THEN
					iCountStop1:=iCountStop1+1;
					IF iCountStop1>iCountStopMax THEN
						iCountStop1:=iCountStopMax+1;
						IF bSearchRight THEN
							iCountDirChange:=2;
						ELSE
							iCountDirChange:=iCountDirChange+1;
						END_IF
						rDirection:=rDirection*(-1);
					END_IF
				ELSE
					iCountStop1:=0;	
				END_IF
				
				//新加的 测试第一阶段搜索正确后不进行第二次搜索
				IF rAGCNow>rAGCInit+rSensitivity THEN
					iCountSearchRight:=iCountSearchRight+1;
				ELSE
					iCountSearchRight:=0;
				END_IF
				IF iCountSearchRight>200 THEN
					iCountSearchRight:=201;
					bSearchRight:=TRUE;
				END_IF
				
			END_IF
		ELSE
			//若是向正走
			IF rCurrentPos>rInterPos THEN
				IF rAGCNow<rAGCMaxValue-rSensitivity THEN
					iCountStop2:=iCountStop2+1;
					IF iCountStop2>iCountStopMax THEN
						iCountStop2:=iCountStopMax+1;
						IF bSearchRight THEN
							iCountDirChange:=2;
						ELSE
							iCountDirChange:=iCountDirChange+1;
						END_IF
						rDirection:=rDirection*(-1);
					END_IF
				ELSE
					iCountStop2:=0;	
				END_IF
				
				//新加的
				IF rAGCNow>rAGCInit+rSensitivity THEN
					iCountSearchRight:=iCountSearchRight+1;
				ELSE
					iCountSearchRight:=0;
				END_IF
				IF iCountSearchRight>200 THEN
					iCountSearchRight:=201;
					bSearchRight:=TRUE;
				END_IF
				
			END_IF
		END_IF
		(*
		IF rAGCNow<rAGCInit-0.05 THEN
			iCountStop1:=iCountStop1+1;
			IF iCountStop1>150 THEN
				iCountDirChange:=iCountDirChange+1;
				rDirection:=rDirection*(-1);
			END_IF
		ELSE
			iCountStop1:=0;	
		END_IF
		*)
		
		 // 记录最强信号的拉偏量和值
		//IF rAGCNow >= rAGCInit AND rAGCNow> rAGCMaxValue THEN
		IF  rAGCNow> rAGCMaxValue THEN
			rAGCMaxBias := rStepBias;
			rAGCMaxValue := rAGCNow;
		END_IF
	END_IF
ELSE
	rStepBias:=0;
	//清空变量
	iCountDirChange:=0;
	rAGCInit:=0;
	rAGCMaxValue:=0;
	rAGCMaxBias:=0;
	rDirection:=1;
	iCountStop1:=0;
	iCountStop2:=0;
	ton(IN:=FALSE,PT:=T#1S,Q=>,ET=>);
	//rStepBias:=0;
	rSearchNextStepTarget:=0;
	bSucess:=FALSE;
	iCountSearchRight:=0;
	bSearchRight:=FALSE;
	iCountBlockEnd:=0;
END_IF


(*
IF rStepBias< rSearchNextStepTarget THEN 
	rStepBias:=rStepBias+rStep;
ELSIF rStepBias> rSearchNextStepTarget THEN
	rStepBias:=rStepBias-rStep;
ELSE
	rStepBias:=rStepBias;
END_IF*)

END_FUNCTION_BLOCK

// Device/Application/扫描搜索/SpiralScan_1
FUNCTION_BLOCK SpiralScan_1
VAR_INPUT
    enable        : BOOL;       // 启动使能
    delta         : REAL;       // 每格步长（°）
    n_steps       : REAL;       // 每格分段周期数
    agc           : REAL;       // 当前AGC
    locked        : BOOL;       // 锁定状态
	AzError       :REAL;
	ELError       :REAL;
END_VAR
VAR_OUTPUT
    azimuth       : REAL;       // 当前方位角输出
    elevation     : REAL;       // 当前俯仰角输出
    done          : BOOL;       // 扫描完成标志
	bType         : BOOL;       // 是否提前结束，1是，0否
END_VAR
VAR
    
    
    lock_count    : INT := 0;
    best_agc      : REAL := 0.0;
    best_az       : REAL := 0.0;
    best_el       : REAL := 0.0;
	bInit         : BOOL;
	icount0       : INT := 0;
	icount1       : INT := 0;
	
	x, y                  : REAL := 0.0;
    dx                	  : REAL := 1.0;
	dy                    : REAL := 0.0;
    step_len              : REAL := 1.0;
    step_count            : REAL := 0.0;
    segment_progress      : REAL := 0.0;
    move_count            : REAL := 1.0;
    state         		  : INT := 0;
    az0, el0              : REAL := 0.0;
    az1, el1              : REAL := 0.0;
    segment_az_step       : REAL := 0.0;
    segment_el_step       : REAL := 0.0;
    side_repeat           : REAL := 0.0;
	icountInit           : INT := 0;
END_VAR


(*==============================================================================
  FB: SpiralScan_1（捕获扫描：螺旋扫描）
  调用者: `SecurityCheck`（段 11），PersistentVars.bSearchType=TRUE 时使用

  与 SpiralScan 区别:
    - 不做矩形格点，而是在网格上按“右→上→左→下”方向逐圈扩展
    - 每一段线性分割为 n_steps 步输出（segment_*_step）
    - 当达到边界条件（az≈4*delta 且 el≈0）或提前锁定即结束

  输出 best_az/best_el:
    - 每拍若 agc 更大，则记录 best_* = -Error（表示需要反向修正误差）
==============================================================================*)
IF NOT enable THEN
    state := 0;
    azimuth := 0.0;
    elevation := 0.0;
    done := FALSE;
	lock_count := 0;
	icount0 := 0;
	segment_progress := 0.0;
	bInit := FALSE;
	best_agc := 0.0;
    best_az := 0.0;
    best_el := 0.0;
	icountInit := 0;
ELSE
    CASE state OF
        // --- 状态0：判断是否已锁定 ---
        0:
			
            
			icountInit := icountInit + 1;
			IF icountInit >= 100 THEN
				icountInit := 101;
				icount0 := icount0 + 1;
				IF locked THEN
					lock_count := lock_count + 1;
				END_IF;
				IF icount0 >= 100 THEN
					IF lock_count >= 10 THEN
						done := TRUE;
						state := 2;   // 提前结束
						lock_count := 0;
					ELSE
						state := 1;   // 转入扫描
						lock_count := 0;
					END_IF;
				END_IF
			END_IF

        // --- 状态1：执行螺旋扫描 ---
        1:
            IF NOT bInit THEN
				x := 0.0; y := 0.0;
				dx := 1.0; dy := 0.0;
				step_len := 1.0;
				step_count := 0.0;
				move_count := 1.0;
				side_repeat := 0.0;
				az0 := 0.0; el0 := 0.0;
				az1 := delta * x;
				el1 := delta * y;
				segment_az_step := (az1 - az0) / n_steps;
				segment_el_step := (el1 - el0) / n_steps;
				segment_progress := 0.0;
				bInit := TRUE;
			ELSE
				
				
				azimuth := az0 + segment_az_step * (segment_progress + 1.0);
				elevation := el0 + segment_el_step * (segment_progress + 1.0);
				segment_progress := segment_progress + 1.0;
				(*
				IF SQRT(azimuth * azimuth + elevation * elevation) > max_radius THEN
						state := 2;
				END_IF
				*)
				
				IF segment_progress >= n_steps THEN
					segment_progress := 0.0;
					az0 := az1;
					el0 := el1;
					// 曼哈顿坐标前进一格
					x := x + dx;
					y := y + dy;
					move_count := move_count + 1.0;
		
					az1 := delta * x;
					el1 := delta * y;
					segment_az_step := (az1 - az0) / n_steps;
					segment_el_step := (el1 - el0) / n_steps;
		
					// 计数并判断是否转弯
					step_count := step_count + 1.0;
					IF step_count >= step_len THEN
						step_count := 0.0;
		
						// 不使用临时变量交换 dx/dy，改为三步法旋转（右→上→左→下）
						IF dx = 1.0 AND dy = 0.0 THEN
							dx := 0.0; dy := 1.0;
						ELSIF dx = 0.0 AND dy = 1.0 THEN
							dx := -1.0; dy := 0.0;
						ELSIF dx = -1.0 AND dy = 0.0 THEN
							dx := 0.0; dy := -1.0;
						ELSIF dx = 0.0 AND dy = -1.0 THEN
							dx := 1.0; dy := 0.0;
						END_IF
		
						side_repeat := side_repeat + 1.0;
						IF side_repeat >= 2.0 THEN
							side_repeat := 0.0;
							step_len := step_len + 1.0;
						END_IF
					END_IF
					
					
				END_IF
				
				IF agc > best_agc THEN
					best_agc := agc;
					best_az := -Azerror;
					best_el := -elError;
				END_IF;
				
				IF ABS(azimuth - 4 * delta) < 1E-6 AND ABS(elevation) < 1E-6 THEN
					state := 3;
				ELSE
					IF locked THEN
					   lock_count := lock_count + 1;
					ELSE
					   lock_count := 0;
					END_IF
					IF lock_count >= 10 THEN
					   done := TRUE;
					   state := 2;   // 提前结束
					   azimuth := best_az;
            		   elevation := best_el;
					END_IF
				END_IF
				
				
			END_IF
        // --- 状态2：提前锁定完成 ---
        2:
            // 保持当前位置即可
            done := TRUE;
			

        // --- 状态3：完成，输出最佳格点 ---
        3:
            azimuth := best_az;
            elevation := best_el;
            done := TRUE;

    END_CASE
	IF state = 3 THEN
		bType := FALSE;
	ELSE
		bType := TRUE;
	END_IF
END_IF;

END_FUNCTION_BLOCK

// Device/Application/Ti_ctrl_1
PROGRAM Ti_ctrl_1

VAR
    Axis3_Ctrl : Ti_Ctrl_FB;           // 倾斜轴控制 FB
    bRemote2LocalStop : BOOL;
    bLocal2RemoteStop : BOOL;
    Error : INT;
    Axis3Limit_pos : REAL;             // +190°
    Axis3Limit_Neg : REAL;             // -190°
    bRTriger : Standard.R_TRIG;
    bFTriger : Standard.F_TRIG;
    Stop3_Count : INT;
    bStop_3 : BOOL;                    // 倾斜轴停稳标志
    rPosModeStepBias : LREAL;
    rPosModeStep : LREAL;
    rStepBiasMax : LREAL;
    rStepBias : LREAL;
    rStep : LREAL;
    rAuToStepBias : LREAL;
    rAutoStep : LREAL;
    TbAutoTrigger : Standard.F_TRIG;
    RbAutoTrigger : Standard.R_TRIG;
    rAutoTrackingBiasMax : LREAL;
    rLocalInitPosModeSpeed : REAL;
    rRemoteInitPosModeSpeed : REAL;
    iCountOffAuto : INT;
    iCasePBAutoTrack : INT;
    rKAuToStepBias : LREAL;
    bVisError : BOOL;                  // 全局错误可视化
END_VAR


(*==============================================================================
  PRG: Ti_ctrl_1（倾斜轴 Ti 顶层程序）
  任务: Canopen 10ms
  作用: 倾斜轴反馈、状态、远/本控切换保护，调用 Ti_Ctrl_FB
  与 El/Az 差异:
    - 无 AGC 搜索、无自跟踪拉偏（相关代码已注释）
    - 未在此程序内赋值 rPIDCmdPos（由 Modbus/其他模块写入后仅做限位）
    - 远控→本控切换时仅强制 Axis3Remote.iMode:=7（本控 mode 未同步置 7）
    - 本控上限钳位有一处写 Axis2Local（原工程保留，勿改）
  软限位: ±190°
==============================================================================*)
IF GVL.Error_code <> 0 THEN
	bVisError := TRUE;
ELSE
	bVisError := FALSE;
END_IF

(* 远控参量注释块为历史 Az 轴拷贝，倾斜轴参数由 Modbus_Slave 写入 Axis3Remote *)

// =============================================================================
// 段 1: 驱动状态 → Axis3Status
// =============================================================================
Axis3Status.Error := GVL.bTiStsBit3;
Axis3Status.ErrorID := GVL.eTiErrorcode;
Axis3Status.bServo_Enable := GVL.bTiStsBit0 AND GVL.bTiStsBit1 AND GVL.bTiStsBit2;
Axis3Status.bBrake := NOT (GVL.bTiStsBit0 AND GVL.bTiStsBit1 AND GVL.bTiStsBit2);
Axis3Status.Disabled := NOT (GVL.bTiStsBit0 AND GVL.bTiStsBit1 AND GVL.bTiStsBit2);
Axis3Remote.rSoft_limit_Negative:=-190;Axis3Remote.rSoft_limit_Postive:=190;
Axis3Local.rSoft_limit_Negative:=-190;Axis3Local.rSoft_limit_Postive:=190;

// =============================================================================
// 段 2: CANopen 反馈 → rFctVelReal_3 / rFctPosReal_3
// =============================================================================
rFctVelReal_3:=DINT_TO_REAL(diTiActVel)/524288.0*360.0;
rFctPosReal_3:=DINT_TO_REAL(diTiActPos)/524288.0*360.0;

// =============================================================================
// 段 3: rPosCmd 硬限位 ±190°
// 注意: 上限分支写的是 Axis2Local（原代码），与 Axis3Local 不一致，保持不改
// =============================================================================
Axis3Limit_pos:=190;
Axis3Limit_Neg:=-190;
IF Axis3Remote.rPosCmd>Axis3Limit_pos THEN
	Axis3Remote.rPosCmd:=190;
ELSIF Axis3Remote.rPosCmd<Axis3Limit_Neg THEN
	 Axis3Remote.rPosCmd:=-190;  
END_IF

IF Axis3Local.rPosCmd>Axis3Limit_pos THEN
	Axis2Local.rPosCmd:=190;
ELSIF Axis3Local.rPosCmd<Axis3Limit_Neg THEN
	 Axis3Local.rPosCmd:=-190;  
END_IF

// =============================================================================
// 段 4: 停稳判定 → Axis3Status.Moving
// =============================================================================
IF  ABS(rFctVelReal_3)<0.035 THEN
	Stop3_Count:=Stop3_Count+1;
	IF Stop3_Count>100 THEN
		Stop3_Count:=101;
		bStop_3:=TRUE;;
	END_IF
ELSE
	Stop3_Count:=0;
	bStop_3:=FALSE;
END_IF
Axis3Status.Moving := NOT bStop_3;

// =============================================================================
// 段 5: PID 使能（mode 2 / 4）
// =============================================================================
IF Axis3Remote.iMode=2 OR Axis3Remote.iMode=4 THEN
	Axis3Remote.bPIDEnable:=TRUE;
ELSE
	Axis3Remote.bPIDEnable:=FALSE;
END_IF

// =============================================================================
// 段 6: 远控 ↔ 本控 切换保护
// 远→本: 仅 Axis3Remote.iMode:=7（与 El/Az 双轴同步 halt 不同）
// =============================================================================
bRTriger(CLK:=GVL.bLocalCtrl);
bFTriger(CLK:=GVL.bLocalCtrl);

IF Axis3Status.bServo_Enable AND (bRTriger.Q ) THEN//如果速度不为0且本控发生切换，则减速停止标识为True
	bRemote2LocalStop:=TRUE;
END_IF
IF bRemote2LocalStop  THEN //若减速停止标识符为True 
	
	IF  bStop_3=TRUE THEN//且电机速度不为0 开始减速 减速完成后下使能，下使能完成后复位标识符复位
		Axis3Local.iMode:=0;
		Axis3Remote.iMode:=0;
		IF Axis3Status.bServo_Enable=FALSE THEN
			bRemote2LocalStop:=FALSE;
		END_IF
	ELSE
		Axis3Remote.iMode:=7;
	END_IF
END_IF

IF Axis3Status.bServo_Enable AND (bFTriger.Q ) THEN//如果速度不为0且本控发生切换，则减速停止标识为True
	bLocal2RemoteStop:=TRUE;
END_IF
IF bLocal2RemoteStop  THEN //若减速停止标识符为True 
	
	IF  bStop_3=TRUE THEN//且电机速度不为0 开始减速 减速完成后下使能，下使能完成后复位标识符复位
		Axis3Local.iMode:=0;
		Axis3Remote.iMode:=0;
		IF Axis3Status.bServo_Enable=FALSE THEN
			bLocal2RemoteStop:=FALSE;
		END_IF
	ELSE
		Axis3Remote.iMode:=7;
		Axis3Local.iMode:=7;
	END_IF
END_IF

(* 自跟踪与 rPIDCmdPos 程引合成在此轴已注释，当前仅对既有 rPIDCmdPos 做限位 *)

// =============================================================================
// 段 7: rPIDCmdPos 限位（赋值在其他 POU，如 Modbus_Slave / RealTimePosCal）
// =============================================================================
IF Axis3Remote.rPIDCmdPos<-190 THEN
	Axis3Remote.rPIDCmdPos:=-190;
ELSIF Axis3Remote.rPIDCmdPos>190 THEN
	Axis3Remote.rPIDCmdPos:=190;
END_IF

Axis3_Ctrl(sLocal:=Axis3Local, sCtrl:=Axis3Remote, sStatus:=Axis3Status, sVisible:=Axis3Visible, rRealPos:=rFctPosReal_3, rPosLimK:=0.34);

END_PROGRAM

// Device/Application/Get_AZ
FUNCTION_BLOCK Get_AZ
VAR_INPUT
	uliRealTime : LREAL; // 当前时间戳，单位毫秒
	lrStartTime : LREAL; // 任务起始时间，单位秒
	rNodeTime1 : REAL;
	rNodeTime2 : REAL;
	rNodeTime3 : REAL;
    rNodeTime4 : REAL;
    rNodeTime5 : REAL;
	rEndTime : REAL;
	lrFun1 : ARRAY[0..10] OF LREAL;
	lrFun2 : ARRAY[0..10] OF LREAL;
	lrFun3 : ARRAY[0..10] OF LREAL;
	lrFun4 : ARRAY[0..10] OF LREAL;
	lrFun5 : ARRAY[0..10] OF LREAL;
	lrFun6 : ARRAY[0..10] OF LREAL;
END_VAR
VAR_OUTPUT
	lrFitResult : LREAL;
END_VAR
VAR
	rDelTime : REAL;
	rRealTime : LREAL;
END_VAR

rRealTime := uliRealTime / 1000.0 - lrStartTime/1000.0;


IF rRealTime <= 0.0 THEN
	rDelTime := 0.0;
	lrFitResult := lrFun1[10];
ELSIF rRealTime <= rNodeTime1 THEN
    rDelTime := rRealTime - 0.0;
	lrFitResult := lrFun1[0] * EXPT(rDelTime,10) + lrFun1[1] * EXPT(rDelTime,9) + lrFun1[2] * EXPT(rDelTime,8) + lrFun1[3] * EXPT(rDelTime,7) + lrFun1[4] * EXPT(rDelTime,6) + lrFun1[5] * EXPT(rDelTime,5)
    + lrFun1[6] * EXPT(rDelTime,4) + lrFun1[7] * EXPT(rDelTime,3) + lrFun1[8] * EXPT(rDelTime,2) + lrFun1[9] * rDelTime + lrFun1[10];
ELSIF rRealTime <= rNodeTime2 THEN
    rDelTime := rRealTime - rNodeTime1;
    lrFitResult := lrFun2[0] * EXPT(rDelTime,10) + lrFun2[1] * EXPT(rDelTime,9) + lrFun2[2] * EXPT(rDelTime,8) + lrFun2[3] * EXPT(rDelTime,7) + lrFun2[4] * EXPT(rDelTime,6) + lrFun2[5] * EXPT(rDelTime,5)
    + lrFun2[6] * EXPT(rDelTime,4) + lrFun2[7] * EXPT(rDelTime,3) + lrFun2[8] * EXPT(rDelTime,2) + lrFun2[9] * rDelTime + lrFun2[10];
ELSIF rRealTime <= rNodeTime3 THEN
    rDelTime := rRealTime - rNodeTime2;
    lrFitResult := lrFun3[0] * EXPT(rDelTime,10) + lrFun3[1] * EXPT(rDelTime,9) + lrFun3[2] * EXPT(rDelTime,8) + lrFun3[3] * EXPT(rDelTime,7) + lrFun3[4] * EXPT(rDelTime,6) + lrFun3[5] * EXPT(rDelTime,5)
    + lrFun3[6] * EXPT(rDelTime,4) + lrFun3[7] * EXPT(rDelTime,3) + lrFun3[8] * EXPT(rDelTime,2) + lrFun3[9] * rDelTime + lrFun3[10];
ELSIF rRealTime <= rNodeTime4 THEN
    rDelTime := rRealTime - rNodeTime3;
    lrFitResult := lrFun4[0] * EXPT(rDelTime,10) + lrFun4[1] * EXPT(rDelTime,9) + lrFun4[2] * EXPT(rDelTime,8) + lrFun4[3] * EXPT(rDelTime,7) + lrFun4[4] * EXPT(rDelTime,6) + lrFun4[5] * EXPT(rDelTime,5)
    + lrFun4[6] * EXPT(rDelTime,4) + lrFun4[7] * EXPT(rDelTime,3) + lrFun4[8] * EXPT(rDelTime,2) + lrFun4[9] * rDelTime + lrFun4[10];
ELSIF rRealTime <= rNodeTime5 THEN
    rDelTime := rRealTime - rNodeTime4;
    lrFitResult := lrFun5[0] * EXPT(rDelTime,10) + lrFun5[1] * EXPT(rDelTime,9) + lrFun5[2] * EXPT(rDelTime,8) + lrFun5[3] * EXPT(rDelTime,7) + lrFun5[4] * EXPT(rDelTime,6) + lrFun5[5] * EXPT(rDelTime,5)
    + lrFun5[6] * EXPT(rDelTime,4) + lrFun5[7] * EXPT(rDelTime,3) + lrFun5[8] * EXPT(rDelTime,2) + lrFun5[9] * rDelTime + lrFun5[10];
ELSIF rRealTime <= rEndTime THEN
    rDelTime := rRealTime - rNodeTime5;
    lrFitResult := lrFun6[0] * EXPT(rDelTime,10) + lrFun6[1] * EXPT(rDelTime,9) + lrFun6[2] * EXPT(rDelTime,8) + lrFun6[3] * EXPT(rDelTime,7) + lrFun6[4] * EXPT(rDelTime,6) + lrFun6[5] * EXPT(rDelTime,5)
    + lrFun6[6] * EXPT(rDelTime,4) + lrFun6[7] * EXPT(rDelTime,3) + lrFun6[8] * EXPT(rDelTime,2) + lrFun6[9] * rDelTime + lrFun6[10];
ELSE
    rDelTime := rEndTime - rNodeTime5;
    lrFitResult := lrFun6[0] * EXPT(rDelTime,10) + lrFun6[1] * EXPT(rDelTime,9) + lrFun6[2] * EXPT(rDelTime,8) + lrFun6[3] * EXPT(rDelTime,7) + lrFun6[4] * EXPT(rDelTime,6) + lrFun6[5] * EXPT(rDelTime,5)
    + lrFun6[6] * EXPT(rDelTime,4) + lrFun6[7] * EXPT(rDelTime,3) + lrFun6[8] * EXPT(rDelTime,2) + lrFun6[9] * rDelTime + lrFun6[10];
END_IF

IF lrFitResult>270 THEN
	lrFitResult:=270;
ELSIF lrFitResult<-270 THEN
	lrFitResult:=-270;
END_IF

END_FUNCTION_BLOCK

// Device/Application/TimeCase
PROGRAM TimeCase
VAR
	stUTC_Timestamp :SYSTIME ;
	stSYS_Timestamp :ULINT ;
	stGNSS_Timestap :ULINT;
    Result : RTS_IEC_RESULT;
	Uptriger:Standard.R_TRIG;
	Triger AT %IX0.0:BOOL;
	Feed AT %QX0.0:BOOL;	
	TON_F: TON;
	dDelPTime: DINT;
	max_DelPTime:DINT :=0; 
	min_DelPTime: DINT :=-999999;
	iCount: INT;
	dtNow: DATE_AND_TIME;
	dtGNSS: DATE_AND_TIME;
	dtLastGNSS: ULINT;
	iDiffETime: DINT;
	DelPTime: DINT;
	
END_VAR

//计算时间误差序列
Result := SysTimeRtcHighResGet(stUTC_Timestamp);        
stSYS_Timestamp := TO_ULINT(stUTC_Timestamp);           // ULINT，获取本地时间
dtNow := TO_DT(stUTC_Timestamp / 1000); 		        // 转换为DATE_AND_TIME类型

Uptriger(CLK:=Triger);                                  //检测PPS上升沿
IF Uptriger.Q THEN                                      //上升沿触发后，GPRMC解析，DO0上升沿输出（电平24V）
	Feed:=TRUE;	
	dtGNSS := TO_DT(GVL.stGNSS_Timestap / 1000); 	    // 拿到串口时间数据			                                     
	iDiffETime:=ULINT_TO_DINT(GVL.stGNSS_Timestap-dtLastGNSS);  
	dtLastGNSS:=GVL.stGNSS_Timestap;                    //缓存上一周期时间戳（ms)  
	dDelPTime:=ULINT_TO_DINT(GVL.stGNSS_Timestap - stSYS_Timestamp);       //计算误差	              
	IF iDiffETime = 1000 THEN                           //确保时间更新步进1S
		IF dDelPTime < 0 THEN                           //更新最小值
			IF dDelPTime < min_DelPTime THEN
				min_DelPTime:=dDelPTime;
				DelPTime:=min_DelPTime;                 
			END_IF		
		ELSE                                            //更新最大值
			IF dDelPTime > max_DelPTime THEN
				max_DelPTime:=dDelPTime;
				DelPTime:=max_DelPTime;
			END_IF
		END_IF	
	END_IF				    						
	iCount:=iCount+1;
	IF iCount >= 60 THEN                                //一分钟校一次时间
		GVL.dDelTime:=DelPTime;
		max_DelPTime:=0;
		min_DelPTime:=0;	
		iCount:=0;
	END_IF
	
END_IF
TON_F(IN:=Feed, PT:=T#100MS, Q=>,ET=>);                 //脉宽200ms（测试时延，为了在示波器看波形）
IF TON_F.Q THEN
	Feed:=FALSE;		
END_IF

END_PROGRAM

// Device/Application/Get_AZ_1
FUNCTION_BLOCK Get_AZ_1
VAR_INPUT
	uliRealTime : LREAL; // 当前时间戳，单位毫秒
	lrStartTime : LREAL; // 任务起始时间，单位秒
	rNodeTime1 : REAL;
	rNodeTime2 : REAL;
	rNodeTime3 : REAL;
    rNodeTime4 : REAL;
    rNodeTime5 : REAL;
	rEndTime : REAL;
	lrFun1 : ARRAY[0..10] OF LREAL;
	lrFun2 : ARRAY[0..10] OF LREAL;
	lrFun3 : ARRAY[0..10] OF LREAL;
	lrFun4 : ARRAY[0..10] OF LREAL;
	lrFun5 : ARRAY[0..10] OF LREAL;
	lrFun6 : ARRAY[0..10] OF LREAL;
END_VAR
VAR_OUTPUT
	lrFitResult : LREAL;
END_VAR
VAR
	rDelTime : REAL;
	rRealTime : LREAL;
END_VAR

rRealTime := uliRealTime / 1000.0 - lrStartTime/1000.0;


IF rRealTime <= 0.0 THEN
	rDelTime := 0.0;
	lrFitResult := lrFun1[10];
ELSIF rRealTime <= rNodeTime1 THEN
    rDelTime := rRealTime - 0.0;
	lrFitResult := lrFun1[0] * EXPT(rDelTime,10) + lrFun1[1] * EXPT(rDelTime,9) + lrFun1[2] * EXPT(rDelTime,8) + lrFun1[3] * EXPT(rDelTime,7) + lrFun1[4] * EXPT(rDelTime,6) + lrFun1[5] * EXPT(rDelTime,5)
    + lrFun1[6] * EXPT(rDelTime,4) + lrFun1[7] * EXPT(rDelTime,3) + lrFun1[8] * EXPT(rDelTime,2) + lrFun1[9] * rDelTime + lrFun1[10];
ELSIF rRealTime <= rNodeTime2 THEN
    rDelTime := rRealTime - rNodeTime1;
    lrFitResult := lrFun2[0] * EXPT(rDelTime,10) + lrFun2[1] * EXPT(rDelTime,9) + lrFun2[2] * EXPT(rDelTime,8) + lrFun2[3] * EXPT(rDelTime,7) + lrFun2[4] * EXPT(rDelTime,6) + lrFun2[5] * EXPT(rDelTime,5)
    + lrFun2[6] * EXPT(rDelTime,4) + lrFun2[7] * EXPT(rDelTime,3) + lrFun2[8] * EXPT(rDelTime,2) + lrFun2[9] * rDelTime + lrFun2[10];
ELSIF rRealTime <= rNodeTime3 THEN
    rDelTime := rRealTime - rNodeTime2;
    lrFitResult := lrFun3[0] * EXPT(rDelTime,10) + lrFun3[1] * EXPT(rDelTime,9) + lrFun3[2] * EXPT(rDelTime,8) + lrFun3[3] * EXPT(rDelTime,7) + lrFun3[4] * EXPT(rDelTime,6) + lrFun3[5] * EXPT(rDelTime,5)
    + lrFun3[6] * EXPT(rDelTime,4) + lrFun3[7] * EXPT(rDelTime,3) + lrFun3[8] * EXPT(rDelTime,2) + lrFun3[9] * rDelTime + lrFun3[10];
ELSIF rRealTime <= rNodeTime4 THEN
    rDelTime := rRealTime - rNodeTime3;
    lrFitResult := lrFun4[0] * EXPT(rDelTime,10) + lrFun4[1] * EXPT(rDelTime,9) + lrFun4[2] * EXPT(rDelTime,8) + lrFun4[3] * EXPT(rDelTime,7) + lrFun4[4] * EXPT(rDelTime,6) + lrFun4[5] * EXPT(rDelTime,5)
    + lrFun4[6] * EXPT(rDelTime,4) + lrFun4[7] * EXPT(rDelTime,3) + lrFun4[8] * EXPT(rDelTime,2) + lrFun4[9] * rDelTime + lrFun4[10];
ELSIF rRealTime <= rNodeTime5 THEN
    rDelTime := rRealTime - rNodeTime4;
    lrFitResult := lrFun5[0] * EXPT(rDelTime,10) + lrFun5[1] * EXPT(rDelTime,9) + lrFun5[2] * EXPT(rDelTime,8) + lrFun5[3] * EXPT(rDelTime,7) + lrFun5[4] * EXPT(rDelTime,6) + lrFun5[5] * EXPT(rDelTime,5)
    + lrFun5[6] * EXPT(rDelTime,4) + lrFun5[7] * EXPT(rDelTime,3) + lrFun5[8] * EXPT(rDelTime,2) + lrFun5[9] * rDelTime + lrFun5[10];
ELSIF rRealTime <= rEndTime THEN
    rDelTime := rRealTime - rNodeTime5;
    lrFitResult := lrFun6[0] * EXPT(rDelTime,10) + lrFun6[1] * EXPT(rDelTime,9) + lrFun6[2] * EXPT(rDelTime,8) + lrFun6[3] * EXPT(rDelTime,7) + lrFun6[4] * EXPT(rDelTime,6) + lrFun6[5] * EXPT(rDelTime,5)
    + lrFun6[6] * EXPT(rDelTime,4) + lrFun6[7] * EXPT(rDelTime,3) + lrFun6[8] * EXPT(rDelTime,2) + lrFun6[9] * rDelTime + lrFun6[10];
ELSE
    rDelTime := rEndTime - rNodeTime5;
    lrFitResult := lrFun6[0] * EXPT(rDelTime,10) + lrFun6[1] * EXPT(rDelTime,9) + lrFun6[2] * EXPT(rDelTime,8) + lrFun6[3] * EXPT(rDelTime,7) + lrFun6[4] * EXPT(rDelTime,6) + lrFun6[5] * EXPT(rDelTime,5)
    + lrFun6[6] * EXPT(rDelTime,4) + lrFun6[7] * EXPT(rDelTime,3) + lrFun6[8] * EXPT(rDelTime,2) + lrFun6[9] * rDelTime + lrFun6[10];
END_IF

IF lrFitResult>90 THEN
	lrFitResult:=90;
ELSIF lrFitResult<3 THEN
	lrFitResult:=3;
END_IF

END_FUNCTION_BLOCK

// Device/Application/插值模块/threesimple2_1
FUNCTION_BLOCK threesimple2_1
VAR_INPUT
	XModbusUL:ARRAY [1..10] OF ULINT:=[1,2,3,4,5,6,7,8,9,10];//输入的Modbus时间数组
	XModbus:ARRAY [1..10] OF LREAL;
	YModbus:ARRAY [1..10] OF LREAL;//输入的Modbus位置数组
	y0:REAL;
	yn:REAL;//y0,yn表示的是S''(x0)=f''(x0)=y0，S''(xn)=f''(xn)=yn,自然边界即条件值为0
	xt:LREAL;//所求目标位置
	
	//bResetErr:BOOL;
END_VAR
VAR_OUTPUT
	sout:REAL;
	nout:INT;
	ErrCode:INT;
	
	bSetZero:BOOL;//Modbus序列清零标识符；
END_VAR
VAR
	Three:three2;
	X:ARRAY [1..5] OF LREAL;
	Y:ARRAY [1..5] OF LREAL;
	
	M :ARRAY [1..5] OF LREAL;
	A: ARRAY [1..5,1..5] OF LREAL;
	D: ARRAY[1..3,1..3] OF LREAL;
	g: ARRAY [1..3] OF LREAL;
	h:ARRAY [1..4] OF LREAL;
	
	n:INT:=5;
	
	p1: ARRAY [1..4] OF REAL;
	p2:ARRAY [1..4] OF REAL;
	p3:ARRAY [1..4] OF REAL;
	p4:ARRAY [1..4] OF REAL;
	i:INT;
	ii:INT;//清空序列
	
	j:INT;//寻找差值区间的循环变量
	k:INT;//插值区间
	iCountOutMaxRange:INT;
	iCountOutMinRange:INT;
	nn:INT;//格式转换循环遍历
	mm:INT;//查重遍历；
END_VAR

FOR nn:=1 TO 10 DO
	//XModbus[nn]:=ULINT_TO_LREAL(XModbusUL[nn])*1000000/1000.0;
	XModbus[nn]:=ULINT_TO_LREAL(XModbusUL[nn]-XModbusUL[1])+1.0;
END_FOR
	xt:=xt-ULINT_TO_LREAL(XModbusUL[1])+1.0;
IF ErrCode>0 THEN
	ErrCode:=0;
END_IF


FOR mm:=2 TO 8 DO
	IF XModbus[mm] = XModbus[mm + 1] THEN
		// 找到相等的两个数，进行线性插值
		XModbus[mm + 1] := (XModbus[mm] + XModbus[mm + 2]) / 2.0;
	END_IF;
END_FOR
IF XModbus[1] = XModbus[2] THEN
	// 找到相等的两个数，进行线性插值
	XModbus[1] := XModbus[2]-(XModbus[3]-XModbus[2]);
END_IF;
IF XModbus[9] = XModbus[10] THEN
	// 找到相等的两个数，进行线性插值
	XModbus[10] := XModbus[9]+(XModbus[9]-XModbus[8]);
END_IF;

IF ErrCode <> 0 THEN
	iCountOutMaxRange:=0;
	iCountOutMinRange:=0;
END_IF


//在何处清空序列呢
//bSetZero:=FALSE; //默认不清空

IF  XModbus[10]=0 THEN
	//报错
	ErrCode:=107;//序列为空
ELSE
	IF XModbus[10]-XModbus[1]>2000000 THEN
		sout:=YModbus[10];
	ELSE
		IF xt<XModbus[1] THEN
			sout:=YModbus[1];
			//报故障 累计超时报错
			iCountOutMinRange:=iCountOutMinRange+1;
			IF iCountOutMinRange>5000 THEN
				iCountOutMaxRange:=5001;
				//ErrCode:=108;//偏小超时报错
			END_IF
		ELSIF xt>XModbus[10]  THEN
			sout:=YModbus[10];
			//报故障 累计超时报错
			iCountOutMaxRange:=iCountOutMaxRange+1;
			IF iCountOutMaxRange>5000 THEN
				iCountOutMaxRange:=5001;
				//ErrCode:=109;//偏大超时报错
			END_IF
		ELSE //若所求目标位置在Modbus中间
			iCountOutMaxRange:=0;
			iCountOutMinRange:=0;
			//若不满五个点
			IF XModbus[6]=0 THEN
				sout:=XModbus[10];
			ELSE
				//若满五个点
				//寻找当前插值区间
				FOR j:=2 TO 10 DO
					IF xt<XModbus[j] THEN
						k:=j;
						EXIT;
					END_IF
				END_FOR
				
				IF k=2 THEN
					X[1]:=XModbus[k-1];X[2]:=XModbus[k];X[3]:=XModbus[k+1];X[4]:=XModbus[k+2];X[5]:=XModbus[k+3];
					y[1]:=YModbus[k-1];Y[2]:=YModbus[k];Y[3]:=YModbus[k+1];Y[4]:=YModbus[k+2];Y[5]:=YModbus[k+3];
				ELSIF k>2 AND k<=8 THEN
					X[1]:=XModbus[k-2];X[2]:=XModbus[k-1];X[3]:=XModbus[k];X[4]:=XModbus[k+1];X[5]:=XModbus[k+2];
					Y[1]:=YModbus[k-2];Y[2]:=YModbus[k-1];Y[3]:=YModbus[k];Y[4]:=YModbus[k+1];Y[5]:=YModbus[k+2];
				ELSIF k=9 THEN
					X[1]:=XModbus[k-3];X[2]:=XModbus[k-2];X[3]:=XModbus[k-1];X[4]:=XModbus[k];X[5]:=XModbus[k+1];
					Y[1]:=YModbus[k-3];Y[2]:=YModbus[k-2];Y[3]:=YModbus[k-1];Y[4]:=YModbus[k];Y[5]:=YModbus[k+1];
				ELSIF k=10 THEN
					X[1]:=XModbus[k-4];X[2]:=XModbus[k-3];X[3]:=XModbus[k-2];X[4]:=XModbus[k-1];X[5]:=XModbus[k];
					Y[1]:=YModbus[k-4];Y[2]:=YModbus[k-3];Y[3]:=YModbus[k-2];Y[4]:=YModbus[k-1];Y[5]:=YModbus[k];
				END_IF
				
				
				//开始解算
				Three(X:=X,Y:=Y,y0:=y0,yn:=yn,D=>D,h=>h,A=>A,g=>g,M=>M);
				FOR i:=1 TO (n-1) DO
					p1[i]:=M[i]*(X[i+1]-xt)*(X[i+1]-xt)*(X[i+1]-xt)/(6*h[i]);
					p2[i]:=M[i+1]*(xt-X[i])*(xt-X[i])*(xt-X[i])/(6*h[i]);
					p3[i]:=(A[i,1]-M[i]/6*(h[i])*(h[i]))*(X[i+1]-xt)/h[i];
					p4[i]:=(A[i+1,1]-M[i+1]/6*(h[i])*(h[i]))*(xt-X[i])/h[i];
				END_FOR
				FOR i:=1 TO (n-1) DO
					IF (xt<=X[i+1])AND (xt>=X[i]) THEN
						nout:=i;
						sout:=p1[nout]+p2[nout]+p3[nout]+p4[nout]; 
					ELSIF xt>X[5] THEN
						nout:=4;
					ELSIF xt<X[1]THEN
						nout:=1;
					END_IF
				END_FOR
				sout:=p1[nout]+p2[nout]+p3[nout]+p4[nout]; 
				(*
				IF xt>X[5] THEN
					nout:=4;
					sout:=p1[nout]+p2[nout]+p3[nout]+p4[nout]; 
				ELSIF xt<X[1] THEN
					nout:=1;
					sout:=p1[nout]+p2[nout]+p3[nout]+p4[nout]; 
				END_IF
				*)
				END_IF
			END_IF
			
		END_IF

//修正输入量为长度为10的数组

END_IF

END_FUNCTION_BLOCK

// Device/Application/插值模块/three2
FUNCTION_BLOCK three2
VAR_INPUT
	X:ARRAY [1..5] OF LREAL;
	Y:ARRAY [1..5] OF LREAL;
	y0:REAL:=0;
	yn:REAL:=0;//y0,yn表示的是S''(x0)=f''(x0)=y0，S''(xn)=f''(xn)=yn,自然边界即条件值为0
END_VAR

VAR_OUTPUT
	M :ARRAY [1..5] OF LREAL;
	A: ARRAY [1..5,1..5] OF LREAL;
	D: ARRAY[1..3,1..3] OF LREAL;
	g: ARRAY [1..3] OF LREAL;
	h:ARRAY [1..4] OF LREAL;
END_VAR

VAR
	n:INT:=5;
	
	
	ypie:ARRAY [1..5] OF REAL;
	j:INT;
	i:INT;
	u :ARRAY [1..3] OF REAL;
	n_: ARRAY [1..3] OF REAL;
	M_:ARRAY [1..3] OF REAL;
	solve:solvex;

	
	iCounttest: INT;
	
	
	miu :ARRAY [1..4] OF REAL;
END_VAR

//此函数为M值求值函数
//D,h,A,g,M输出量分别为系数矩阵D，插值宽度h，差商表A，g值,M值 
n:=5;
//A(:,1)=Y'
A[1,1]:=Y[1];A[2,1]:=Y[2];A[3,1]:=Y[3];A[4,1]:=Y[4];A[5,1]:=Y[5];

//A(:,1)=Y'
FOR j :=2 TO 5 DO
	FOR i:=j TO 5 DO
		A[i,j]:=(A[i,j-1]- A[i-1,j-1])/(X[i]-X[i-j+1]);
	END_FOR
END_FOR


FOR i:=1 TO (n-1) DO
	h[i]:=X[i+1]-X[i];
END_FOR


//h[1]:=X[2]-X[1];h[2]:=X[3]-X[2];h[3]:=X[4]-X[3];h[4]:=X[5]-X[4];



//D[1,1]:=2;D[2,2]:=2;D[3,3]:=2;

FOR i:=1 TO n-2 DO
	D[i,i]:=2; 
	IF i=1 THEN
		g[i]:=(6/(h[i+1]+h[i]))*(A[i+2,2]-A[i+1,2])-h[i]/(h[i]+h[i+1])*y0;
	ELSIF i=(n-2) THEN
		g[i]:=(6/(h[i+1]+h[i]))*(A[i+2,2]-A[i+1,2])-(1-h[i]/(h[i]+h[i+1]))*yn;
	ELSE
		g[i]:=(6/(h[i+1]+h[i]))*(A[i+2,2]-A[i+1,2]);
	END_IF
END_FOR



FOR i:=2 TO (n-2) DO
	u[i]:=h[i]/(h[i]+h[i+1]);
	n_[i-1]:=h[i]/(h[i-1]+h[i]);
	D[i-1,i]:=n_[i-1];
	D[i,i-1]:=u[i];
END_FOR


solve(M:=D,G:=g,X=>M_);
M[1]:=0;M[5]:=0;M[2]:=M_[1];M[3]:=M_[2];M[4]:=M_[3];

END_FUNCTION_BLOCK

// Device/Application/插值模块/solvex
FUNCTION_BLOCK solvex

VAR_IN_OUT
	M: ARRAY [1..3, 1..3] OF LREAL ; // 定义3x3矩阵M
    G: ARRAY [1..3] OF LREAL ; // 定义3x1数组G
END_VAR
VAR
    
   
	AdjointMatrix: ARRAY [1..3, 1..3] OF REAL; // 用于存储伴随矩阵
	Determinant: REAL; //行列式
    //M_Inverse: ARRAY [1..3, 1..3] OF REAL; //逆矩阵
    i, j, k: INT;
    Temp: REAL;

   

END_VAR

VAR_OUTPUT
	X: ARRAY [1..3] OF REAL; // 用于存储解x
END_VAR


// 计算矩阵的行列式
Determinant := M[1, 1] * (M[2, 2] * M[3, 3] - M[2, 3] * M[3, 2]) -
               M[1, 2] * (M[2, 1] * M[3, 3] - M[2, 3] * M[3, 1]) +
               M[1, 3] * (M[2, 1] * M[3, 2] - M[2, 2] * M[3, 1]);

(*
// 计算3x3矩阵的伴随矩阵
Determinant := M[1, 1] * (M[2, 2] * M[3, 3] - M[2, 3] * M[3, 2]) -
               M[1, 2] * (M[2, 1] * M[3, 3] - M[2, 3] * M[3, 1]) +
               M[1, 3] * (M[2, 1] * M[3, 2] - M[2, 2] * M[3, 1]);

IF ABS(Determinant) > 1.0E-6 THEN
    FOR i := 1 TO 3 DO
        FOR j := 1 TO 3 DO
            AdjointMatrix[i, j] := M[(i MOD 3) + 1, (j MOD 3) + 1] * M[((i + 1) MOD 3) + 1, ((j + 1) MOD 3) + 1] -
                                   M[(i MOD 3) + 1, ((j + 1) MOD 3) + 1] * M[((i + 1) MOD 3) + 1, (j MOD 3) + 1];
        END_FOR
    END_FOR

    FOR i := 1 TO 3 DO
        FOR j := 1 TO 3 DO
            AdjointMatrix[j, i] := AdjointMatrix[i, j];
            AdjointMatrix[i, j] := AdjointMatrix[i, j] / Determinant;
        END_FOR
    END_FOR
END_IF
*)
// 计算3x3矩阵的伴随矩阵
Determinant := M[1, 1] * (M[2, 2] * M[3, 3] - M[2, 3] * M[3, 2]) -
               M[1, 2] * (M[2, 1] * M[3, 3] - M[2, 3] * M[3, 1]) +
               M[1, 3] * (M[2, 1] * M[3, 2] - M[2, 2] * M[3, 1]);

IF ABS(Determinant) > 1.0E-6 THEN
    FOR i := 1 TO 3 DO
        FOR j := 1 TO 3 DO
            AdjointMatrix[j, i] := ((M[(i MOD 3) + 1, (j MOD 3) + 1] * M[((i + 1) MOD 3) + 1, ((j + 1) MOD 3) + 1] -
                                   M[(i MOD 3) + 1, ((j + 1) MOD 3) + 1] * M[((i + 1) MOD 3) + 1, (j MOD 3) + 1]) / Determinant);
        END_FOR
    END_FOR
END_IF

// 计算X = AdjointMatrix * G
FOR i := 1 TO 3 DO
    X[i] := 0.0;
    FOR j := 1 TO 3 DO
        X[i] := X[i] + AdjointMatrix[i, j] * G[j];
    END_FOR
END_FOR

END_FUNCTION_BLOCK

// Device/Application/GetACUTime
PROGRAM GetACUTime
VAR
    tp      : TP;           // 脉冲定时器
    toggle  : BOOL := FALSE; // 当前输出状态
    clk     : BOOL := FALSE; // 方波输出
    tick_ms : TIME := T#500MS; // 高电平/低电平持续时间
	Result : RTS_IEC_RESULT;
	stUTC_Timestamp :SYSTIME ;
	
	dRTime:ULINT;//上位机外部时间 单位ns Unix时间戳，起点是1970-1-1 0:0:0
	dModbusTime:ULINT;//Modbus临时外部时间
	iCountRemote:INT; //上位机锁定判断时间常数
	dCountRemote:ULINT;//上位机时间滑动平均常数
	dLastRTime:ULINT;//上位机上一次外部时间 单位ns Unix时间戳，起点是1970-1-1 0:0:0
	iDiffRTime:DINT;//上位机时间差值
	dDelRTime:LINT;
	dMeanDelRTime:LINT;
	rTriger:Standard.R_TRIG;//上升沿触发器
	
	iDiff:DINT;//实际时间差值
	iDiffLocal:DINT;//本地时间差值
	iDiffETime:DINT;//外部时间差值
	ulACUTimeStamp : ULINT;
END_VAR


// 每次TP结束时翻转状态
IF NOT tp.Q THEN
    toggle := NOT toggle;
    tp.IN := TRUE;
    tp.PT := tick_ms;
ELSE
    tp.IN := FALSE;
END_IF

tp();

Result := SysTimeRtcHighResGet(stUTC_Timestamp);
rTriger(CLK:=toggle);
IF rTriger.Q THEN
	dRTime := modbus_slave.UTC_New;
	iDiffRTime:=ULINT_TO_DINT(dRTime-dLastRTime);
	IF ABS(iDiffRTime)>500 THEN //两次PTP时间差如果大于500毫秒,则判断为上位机时间失锁
		iCountRemote:=0;
		dCountRemote:=0;
		GVL.bRemoteTimeLock:=FALSE;
	ELSE//否则判断为上位机时间锁定并累计1分钟
		iCountRemote:=iCountRemote+1;
	END_IF
	
